# B&R Automation Studio project 8238 (part 5)

#### custom.st
```iecst
PROGRAM _INIT

	Std.TestMode;

//	FOR n := 1 TO MAX_CONTACTRON DO
//		incline						ACCESS ADR(IO_Link.Contactron[n]);
//		incline.Cmd.Reset_Automatic		:= 1;
//		tripCurrent						:= CONTACTRON_TRIP_50_PERCENT;
//		//tripCurrent						:= CONTACTRON_TRIP_75_PERCENT;
//	END_FOR;
//
//	camera ACCESS ADR(Camera[1].Interface);
//
//	gSettings.Drive[1].MotorSize	 			:= ABB_MOTOR_0_75KW;
//	gSettings.Drive[2].MotorSize	 			:= ABB_MOTOR_0_75KW;
//	gSettings.Drive[3].MotorSize	 			:= ABB_MOTOR_3KW;
//	gSettings.Drive[4].MotorSize	 			:= ABB_MOTOR_3KW;
////	gSettings.Drive[3].MotorSize	 			:= ABB_MOTOR_CUSTOM; //from motor template
//
//	FOR n := 1 TO MAX_DRIVES DO
//		ABB_EPL.Drives[n].Cmd.Direction 		:= ABB_DIRECTION_FWD;
//		ABB_EPL.Drives[n].Cmd.TargetVelocity 	:= gSettings.Drive[n].TargetVelocity;
//		gSettings.Drive[n].AccTime 				:= 0.5;
//		gSettings.Drive[n].DecTime 				:= 0.2;
//		gSettings.Drive[n].BrakeFitted			:= 0;
//	END_FOR;

END_PROGRAM

PROGRAM _CYCLIC

//	//==============================
//	//Inclines
//	//==============================
//
//	FOR n := 1 TO MAX_CONTACTRON DO
//		incline					ACCESS ADR(IO_Link.Contactron[n]);
//		IF 	(incline.Comms.Read.CurrentStatus = 0) THEN
//			incline.Cmd.Current		:= tripCurrent;
//		END_IF;
//	END_FOR;
//
//	IO_Link.Contactron[1].Cmd.Run := r57.run_slant; //SICU1		//Y[1399].Y06
//	IO_Link.Contactron[2].Cmd.Run := r116.run_slant; //CICU1
//	IO_Link.Contactron[3].Cmd.Run := r101.run_slant; //CICU2
//	IO_Link.Contactron[4].Cmd.Run := r127.run_slant; //CICU3
////	IO_Link.Contactron[2].Cmd.Run := r21.run_slant; //CICU4
//
//	//====================================
//	//TRN Controls
//	//====================================
//
//	//STRN2
//	r62.request_rotate := (r25.state = 1) AND (OpcUa.VC[232].Read.PositionNo = 2) AND (OpcUa.VC[232].Read.Auto) AND (OpcUa.VC[232].Read.ReadyToReceive) AND NOT r25.safety_zone;
//	ton_rotated_strn2(IN:= (r62.sw_out_a AND r62.sw_out_b),PT := T#2s);
//	ton_straight_strn2(IN:= (r62.sw_in_a AND r62.sw_in_b),PT := T#2s);
//	r62.custom_bring_lock := ton_rotated_strn2.Q OR r62.front_a OR r62.front_b OR NOT r62.rail_mt;
//	rotate_r62 := ((r62.state >= 6) AND (r62.state <= 7)) OR (r62.state = 9);
//	straight_r62 := ((r62.state = 8) OR (r62.state = 1) OR (r62.state = 5));
//	r62.clamp := (rotate_r62 AND NOT ton_rotated_strn2.Q) OR (straight_r62 AND NOT ton_straight_strn2.Q);  // We have to fire this to unlock the rails so we can move them
//
//	r25.custom_bring_lock := NOT ton_rotated_strn2.Q;
//	//r63.custom_bring_lock := NOT ton_straight_strn2.Q;
//
//	//STRN1
//	r63.request_rotate := NOT r22.safety_zone;
//	ton_rotated_strn1(IN:= (r63.sw_out_a AND r63.sw_out_b),PT := T#2s);
//	ton_straight_strn1(IN:= (r63.sw_in_a AND r63.sw_in_b),PT := T#2s);
//	r63.custom_bring_lock := ton_rotated_strn2.Q OR r63.front_a OR r63.front_b OR NOT r63.rail_mt OR NOT ton_straight_strn2.Q;
//	rotate_r63 := ((r63.state >= 6) AND (r63.state <= 7)) OR (r63.state = 9);
//	straight_r63 := ((r63.state = 8) OR (r63.state = 1) OR (r63.state = 5));
//	r63.clamp := (rotate_r63 AND NOT ton_rotated_strn1.Q) OR (straight_r63 AND NOT ton_straight_strn1.Q);  // We have to fire this to unlock the rails so we can move them
//
//	r22.custom_bring_lock := NOT ton_rotated_strn1.Q;
//
//
//	//CTRN1
//	r135.request_rotate := (r65.state = 1) AND (OpcUa.VC[241].Read.PositionNo = 2) AND (OpcUa.VC[241].Read.Auto) AND (OpcUa.VC[241].Read.ReadyToReceive);
//	ton_rotated_ctrn1(IN:= (r135.sw_out_a AND r135.sw_out_b), PT := T#2s);
//	ton_straight_ctrn1(IN:= (r135.sw_in_a AND r135.sw_in_b), PT := T#2s);
//	r135.custom_bring_lock := ton_rotated_ctrn1.Q OR r135.front_a OR r135.front_b OR NOT r135.rail_mt;
//	rotate_r135 := ((r135.state >= 6) AND (r135.state <= 7)) OR (r135.state = 9);
//	straight_r135 := ((r135.state = 8) OR (r135.state = 1) OR (r135.state = 5));
//	r135.clamp := (rotate_r135 AND NOT ton_rotated_ctrn1.Q) OR (straight_r135 AND NOT ton_straight_ctrn1.Q);  // We have to fire this to unlock the rails so we can move them
//
//	//CTRN2
//	r133.request_rotate := (r68.state = 1) AND (OpcUa.VC[242].Read.PositionNo = 2) AND (OpcUa.VC[242].Read.Auto) AND (OpcUa.VC[242].Read.ReadyToReceive);
//	ton_rotated_ctrn2(IN:= (r133.sw_out_a AND r133.sw_out_b), PT := T#2s);
//	ton_straight_ctrn2(IN:= (r133.sw_in_a AND r133.sw_in_b), PT := T#2s);
//	r133.custom_bring_lock := ton_rotated_ctrn2.Q OR r133.front_a OR r133.front_b OR NOT r133.rail_mt;
//	rotate_r133 := ((r133.state >= 6) AND (r133.state <= 7)) OR (r133.state = 9);
//	straight_r133 := ((r133.state = 8) OR (r133.state = 1) OR (r133.state = 5));
//	r133.clamp := (rotate_r133 AND NOT ton_rotated_ctrn2.Q) OR (straight_r133 AND NOT ton_straight_ctrn2.Q);  // We have to fire this to unlock the rails so we can move them
//
//
////	//====================================
////	//TRF Controls
////	//====================================
////
////	ton_clear_strf1(IN:= (NOT r22.front_a AND NOT r22.front_b),PT := T#2s);
////	ton_clear_strf2(IN:= (NOT r25.front_a AND NOT r25.front_b),PT := T#2s);
////
////	r63.custom_send_lock	:=	NOT ton_clear_strf1.Q AND (r22.state >= 5);
////	r62.custom_send_lock	:=	NOT ton_clear_strf2.Q AND (r25.state >= 5);
//
////==============================
////Custom for CDC6 & CDC7
////==============================
//	RequestBag 		:= WORD_TO_INT(plc_info1);
//	IF RequestBag = 7 THEN
//		cdc7RequestBag := TRUE;
//		cdc6RequestBag := FALSE;
//	ELSIF RequestBag = 6 THEN
//		cdc6RequestBag := TRUE;
//		cdc7RequestBag := FALSE;
//	ELSE
//		cdc6RequestBag := FALSE;
//		cdc7RequestBag := FALSE;
//	END_IF;
//
//	r104.lift_stp := r106.going_to;
//
//	// Clean custom code
//	r104.custom_bring_lock := cdc7RequestBag OR r106.going_to;
//	r106.custom_bring_lock := r104.going_to OR r104.front_raw OR NOT r104.rail_mt OR r104.fire;
//
//	r104.going_to;
//	r106.going_to;
//	r103.custom_send_lock;
////==============================
////Sorting Stations Mapping
////==============================
//
////	r41.jogmode := 1;	//set belt pulse mode = TRUE
////	r42.jogmode := 1;
////	r43.jogmode := 1;
////	r44.jogmode := 1;
////	r45.jogmode := 1;
////	r46.jogmode := 1;
////	r47.jogmode := 1;
////	r48.jogmode := 1;
////	r49.jogmode := 1;
////	r50.jogmode := 1;
//
//	//	IO_Link.Contactron[2].Cmd.Run := r41.run_conveyor AND (r40.conveyor_running OR (r40.run_conveyor AND Std.TestMode));
//	//	IO_Link.Contactron[3].Cmd.Run := r42.run_conveyor AND (r40.conveyor_running OR (r40.run_conveyor AND Std.TestMode));
//	//	IO_Link.Contactron[4].Cmd.Run := r43.run_conveyor AND (r40.conveyor_running OR (r40.run_conveyor AND Std.TestMode));
//	//	IO_Link.Contactron[5].Cmd.Run := r44.run_conveyor AND (r40.conveyor_running OR (r40.run_conveyor AND Std.TestMode));
//	//	IO_Link.Contactron[6].Cmd.Run := r45.run_conveyor AND (r40.conveyor_running OR (r40.run_conveyor AND Std.TestMode));
//	//	IO_Link.Contactron[7].Cmd.Run := r46.run_conveyor AND (r40.conveyor_running OR (r40.run_conveyor AND Std.TestMode));
//	//	IO_Link.Contactron[8].Cmd.Run := r47.run_conveyor AND (r40.conveyor_running OR (r40.run_conveyor AND Std.TestMode));
//	//	IO_Link.Contactron[9].Cmd.Run := r48.run_conveyor AND (r40.conveyor_running OR (r40.run_conveyor AND Std.TestMode));
//	//	IO_Link.Contactron[10].Cmd.Run := r49.run_conveyor AND (r40.conveyor_running OR (r40.run_conveyor AND Std.TestMode));
//	//	IO_Link.Contactron[11].Cmd.Run := r50.run_conveyor AND (r40.conveyor_running OR (r40.run_conveyor AND Std.TestMode));
//	//
//	r1.custom_send_lock := r1.over_weight;
//	r2.custom_send_lock := r2.over_weight;
//	r3.custom_send_lock := r3.over_weight;
//	r4.custom_send_lock := r4.over_weight;
//	r5.custom_send_lock := r5.over_weight;
//	r6.custom_send_lock := r6.over_weight;
//	r7.custom_send_lock := r7.over_weight;
//	r8.custom_send_lock := r8.over_weight;
//	r9.custom_send_lock := r9.over_weight;
//	r10.custom_send_lock := r10.over_weight;
//	r11.custom_send_lock := r11.over_weight;
//	r12.custom_send_lock := r12.over_weight;
//	r13.custom_send_lock := r13.over_weight;
//	r14.custom_send_lock := r14.over_weight;
//	r15.custom_send_lock := r15.over_weight;
//	r16.custom_send_lock := r16.over_weight;
//	r17.custom_send_lock := r17.over_weight;
//	r18.custom_send_lock := r18.over_weight;
//	r19.custom_send_lock := r19.over_weight;
//	r20.custom_send_lock := r20.over_weight;
//
//	//==============================
//	//Speed Reducers
//	//==============================
//
//	////////////////////////SSR1 is a brush style//////////////////////////
//
//	//inputs
//	i_bagApproach[1] := ssr1_prs; //ssr1 on soiled system
//	//i_bagApproach[2] := ssr2_prs; //ssr2 on soiled system
//	//i_bagApproach[3] := csr1_prs; //csr1 on clean system
//
//	FOR n := 1 TO MAX_SPEED_REDUCERS DO
//
//		ctu_tripCount[n](CU := i_bagApproach[n],PV := 2,RESET := ton_10ms_openBrush[n].Q);
//		ton_10ms_openBrush[n](IN := NOT SafetyZone[1].HaltSys AND o_closeBrush[n], PT := 300);
//
//		IF (ctu_tripCount[n].CV >= 2) THEN
//			o_closeBrush[n] := TRUE;
//		END_IF;
//
//		IF ton_10ms_openBrush[n].Q THEN
//			o_closeBrush[n] := FALSE;
//		END_IF;
//	END_FOR;
//
//	//Outputs
//	ssr1_close := o_closeBrush[1];
////	ssr2_close := o_closeBrush[2];
////	csr1_close := o_closeBrush[3];
//
//
//
//	//==============================
//	//ABB DRIVES
//	//==============================
//
//	FOR n := 1 TO MAX_DRIVES DO
//		ABB_EPL.Drives[n].Cmd.TargetVelocity := gSettings.Drive[n].TargetVelocity;
//	END_FOR;
//
//	ABB_EPL.Drives[1].Cmd.QuickStop := NOT SafetyZone[1].HaltSys; //SB1
//	ABB_EPL.Drives[2].Cmd.QuickStop := NOT SafetyZone[1].HaltSys; //SB2
//	ABB_EPL.Drives[3].Cmd.QuickStop := NOT SafetyZone[4].HaltSys; //STB1
//	ABB_EPL.Drives[4].Cmd.QuickStop := NOT SafetyZone[5].HaltSys; //STB2
//
////	tof_largeload(IN := X[1351].X06, PT:=t#10s);
////	IF tof_largeload.Q THEN
////		ABB_EPL.Drives[2].Cmd.TargetVelocity := gSettings.Drive[2].TargetVelocity/2;
////		//testspeed := gSettings.Drive[2].TargetVelocity/2;
////	ELSE
////		ABB_EPL.Drives[2].Cmd.TargetVelocity := gSettings.Drive[2].TargetVelocity;
////		//testspeed := gSettings.Drive[2].TargetVelocity;
////	END_IF;
//
//	//==============================
//	//SB1 & SB2 - PB control
//	//==============================
//	IF EDGENEG (sb1_start) THEN
//		runBelts_SB1 := 1;
//	END_IF;
//	IF NOT sb1_stop OR SafetyZone[1].HaltSys THEN
//		runBelts_SB1 := 0;
//	END_IF;
//
//	IF EDGENEG (sb2_start) THEN
//		runBelts_SB2 := 1;
//	END_IF;
//	IF NOT sb2_stop OR SafetyZone[1].HaltSys THEN
//		runBelts_SB2 := 0;
//	END_IF;
//
//	sb1_lamp := runBelts_SB1;
//	sb2_lamp := runBelts_SB2;
//
//	ABB_EPL.Drives[1].Cmd.Run := (runBelts_SB1) AND sb1_endPX;
//	ABB_EPL.Drives[2].Cmd.Run := (runBelts_SB2) AND sb2_endPX;
//	ABB_EPL.Drives[3].Cmd.Run := r21.run_conveyor;
//	r21.conveyor_running := ABB_EPL.Drives[3].Status.Running OR r21.run_conveyor;
//	ABB_EPL.Drives[4].Cmd.Run := r24.run_conveyor;
//	r24.conveyor_running := ABB_EPL.Drives[4].Status.Running OR r24.run_conveyor;
//
//
//	//==============================
//	//UI Indicators - in iolist
//	//==============================
//
//
//
//	//==============================
//	//Timers
//	//==============================
//
//	SetValueByName('R043','DBNC_after_time',50);
//	SetValueByName('R045','DBNC_after_time',50);
//	SetValueByName('R047','DBNC_after_time',50);
//	SetValueByName('R092','DBNC_after_time',50);
////	SetValueByName('R047','DBNC_after_time',50);
////	SetValueByName('R047','DBNC_after_time',50);
//	//	SetValueByName('R042','PulseTimerOffTime',1000);
////	//SetValueByName('R043','PulseTimerOnTime',3000);
////	SetValueByName('R043','PulseTimerOffTime',1000);
////	//SetValueByName('R044','PulseTimerOnTime',3000);
////	SetValueByName('R044','PulseTimerOffTime',1000);
////	//SetValueByName('R045','PulseTimerOnTime',3000);
////	SetValueByName('R045','PulseTimerOffTime',1000);
////	//SetValueByName('R046','PulseTimerOnTime',3000);
////	SetValueByName('R046','PulseTimerOffTime',1000);
////	//SetValueByName('R047','PulseTimerOnTime',3000);
////	SetValueByName('R047','PulseTimerOffTime',1000);
////	//SetValueByName('R048','PulseTimerOnTime',3000);
////	SetValueByName('R048','PulseTimerOffTime',1000);
////	//SetValueByName('R049','PulseTimerOnTime',3000);
////	SetValueByName('R049','PulseTimerOffTime',1000);
////	//SetValueByName('R050','PulseTimerOnTime',3000);
////	SetValueByName('R050','PulseTimerOffTime',1000);
////	//SetValueByName('R041','PulseTimerOnTime',3000);
////	//SetValueByName('R041','PulseTimerOffTime',5000);
////	//SetValueByName('R040','MaximumRunningTime',200000);
////	//	SetValueByName('R041','DBNC_front_time',2000);
////	//	SetValueByName('R076','DBNC_front_time',1000);
////	//
////
////	// Camera
////	camera.Read := r31.front;
////	IF camera.ResultReady AND r31.front THEN
////		brsmemcpy(ADR(barcode1),ADR(camera.Result),SIZEOF(barcode1));
////	ELSE
////		brsmemset(ADR(barcode1),0,SIZEOF(barcode1));
////	END_IF;
////
////	IF EDGEPOS(camera.Read) THEN
////		readCount := readCount + 1;
////	END_IF;
////
////
////	//
////	tof_cameraClean(IN := (readCount > 100), PT:=t#2s);
////	r31.puncher := NOT tof_cameraClean.Q;
////
////	IF (readCount > 105) THEN
////		readCount := 0;
////	END_IF;

END_PROGRAM
```

#### Variables.var
```iecst
VAR
	incline : REFERENCE TO Contactron_Type;
	ton_settled : TON_10ms;
	ton_tiltDown : TON_10ms;
	ton_tiltUp : TON_10ms;
	ton_CloserDown : TON_10ms;
	ton_CloserUp : TON_10ms;
	tilt : USINT;
	ton_WaitExtendArm : TON_10ms;
	n : USINT;
	recircLoad : BOOL;
	runBelts : BOOL;
	CarousalBlockedTime : UDINT;
	CarousalBlockedTimer : TON_10ms;
	tof_pressure_1 : TOF;
	tof_open_pressure_1 : TOF;
	camera : REFERENCE TO Camera_interface_typ;
	testing : BOOL;
	testweight1 : UINT;
	testweight2 : UINT;
	runBelts_SB1 : BOOL;
	runBelts_SB2 : BOOL;
	tof_cameraClean : TOF;
	readCount : UINT;
	r81_clear_timer : TON;
	clear_time : UDINT := 5000;
	tof_pressureTime : UDINT := 3000;
	tof_pressureTime2 : UDINT := 1000;
	ctu_tripCount : ARRAY[0..MAX_SPEED_REDUCERS] OF CTU;
	i_bagApproach : ARRAY[0..MAX_SPEED_REDUCERS] OF BOOL;
	ton_10ms_countDebounce : ARRAY[0..MAX_STATIONS] OF TON_10ms;
	ton_10ms_openBrush : ARRAY[0..MAX_SPEED_REDUCERS] OF TON_10ms;
	o_closeBrush : ARRAY[0..MAX_SPEED_REDUCERS] OF BOOL;
	lowerGuard : BOOL;
	tof_largeload : TOF;
	testspeed : INT;
	ton_rotated_strn1 : TON;
	ton_straight_strn1 : TON;
	ton_rotated_strn2 : TON;
	ton_straight_strn2 : TON;
	ton_clear_strf1 : TON;
	ton_clear_strf2 : TON;
	rotate_r62 : BOOL;
	straight_r62 : BOOL;
	rotate_r63 : BOOL;
	straight_r63 : BOOL;
	ton_rotated_ctrn1 : TON;
	ton_straight_ctrn1 : TON;
	ton_rotated_ctrn2 : TON;
	ton_straight_ctrn2 : TON;
	ton_clear_ctrf1 : TON;
	ton_clear_ctrf2 : TON;
	rotate_r135 : BOOL;
	straight_r135 : BOOL;
	rotate_r133 : BOOL;
	straight_r133 : BOOL;
	RequestBag : INT;
	countMode : BOOL;
	iCount : ARRAY[0..MAX_STATIONS] OF BOOL;
	cntDebounceLatch : ARRAY[0..MAX_STATIONS] OF BOOL;
END_VAR
```

#### LocalFunctions.fun
```iecst
{REDUND_ERROR} FUNCTION SetValueByName : BOOL (**Set Local variable from external task*) (*$GROUP=User,$CAT=User,$GROUPICON=User.png,$CATICON=User.png*)
	VAR_INPUT
		TaskName : STRING[24];
		VarName : STRING[50];
		Value : UDINT;
	END_VAR
	VAR
		sVar : UDINT;
		pVar : UDINT;
		varName : STRING[75];
	END_VAR
END_FUNCTION
```

#### SetValueByName.st
```iecst
//*Set Local variable from external task
FUNCTION SetValueByName
	SetValueByName := 0;
	varName := '::';
	brsstrcat(ADR(varName),ADR(TaskName));
	brsstrcat(ADR(varName),ADR(':'));
	brsstrcat(ADR(varName),ADR(VarName));

	IF (PV_xgetadr(ADR(varName),ADR(pVar),ADR(sVar)) = 0) THEN
		IF (SIZEOF(Value) <= sVar)THEN
			brsmemcpy(pVar,ADR(Value),SIZEOF(Value));
			SetValueByName := 1;
		ELSE
			brsmemcpy(pVar,ADR(Value),sVar);
			SetValueByName := 1;
		END_IF;
	END_IF;
END_FUNCTION
```

- Visualisation Logical/mappView (not shown)

### SystemConstants.var - *SYSTEM Constants
```iecst
VAR CONSTANT
	MAX_CAMERAS : USINT := 1; (** Number of B&R Barcode scanners*)
	MAX_SPEED_REDUCERS : USINT := 1; (*Set to number of speed reducers*)
	MAX_CONTACTRON : USINT := 4;
	MAX_DRIVES : USINT := 16; (*Set to number of drives*)
	MAX_FUSE_BANKS : USINT := 11;
	MAX_DUAL_CHANNELS : USINT := 10; (** Number of Estops*)
	MAX_HOIST : USINT := 4;
	MAX_SAFE_ZONES : USINT := 30;
	MAX_RAILS : UINT := 136; (**DO NOT USE -> USE RAIL_COUNT INSTEAD*)
END_VAR
```

### Program Logical/Standard/Program (IEC) - * PLAY AREA

#### Variables.var
```iecst
VAR
	myBuffer : ARRAY[0..511] OF INT;
	myAsIoTrcGet : AsIoTrcGet;
	mO_info : MO_info;
	test : UINT;
	datObjCreate : DatObjCreate;
	FileCreate_0 : FileCreate;
	FileInfo_0 : FileInfo;
	FileOpen_0 : FileOpen;
	ident : UDINT;
	Path : STRING[80];
	fileRW : fileReadWrite;
	sysFileName : STRING[10];
	getModuleName : GetModuleName;
	moduleAddress : STRING[30];
	testUsint : USINT;
END_VAR
```

#### Main.st
```iecst
PROGRAM _INIT
	(* Insert code here *)
	Path := 'SL1.IF1.ST11.IF1.ST3.TRC';
	myAsIoTrcGet.pDevice := ADR(Path);//'SS1.IF1.ST131.TRC');
	myAsIoTrcGet.pBuffer := ADR(myBuffer);
	myAsIoTrcGet.bufferLen := SIZEOF(myBuffer);
	//Sys file to try
//	User			XML - Users
//	Role			XML - Roles
//	sysconf			NOT AVAILABLE ?
//	ashwd			NOT READABLE
//	arconfig		XML -- Contains all hardware configuration  !!! Use this to get module name. ***
//	asfw			NOT READABLE
//	ashwac			XML -- No data ??
//	iomap			IO File - Readable
//	asiol1			XML -- No data ??
//	asiol3			XML -- No data ??
//	Config			XML -- MAPP Components config
//	TC				XML -- Text Config.
//	viComp			VISION
//	Settings		VISION
//	viAppBCDE		VISION

	sysFileName := 'iomap';
END_PROGRAM

PROGRAM _CYCLIC

	//We can run an IO trace.. Is this useful when looking for breaks in the IO.. Maybe we can run somekind of automated test.

	IF myAsIoTrcGet.enable <> 0 THEN
		myAsIoTrcGet();
		myAsIoTrcGet.enable := 0;
	END_IF

	// Testing resolving the Module Name.

	CASE test OF
		10:

			mO_info(enable := 1, pName := ADR(sysFileName), grp := 0);
			IF mO_info.status = ERR_OK THEN
				test := 20;
			END_IF;

		20:// File Write
			fileRW.enable := 1;
			fileRW.mode := FILE_SAVE;
			fileRW.pData := mO_info.address;
			fileRW.sizeData := 	mO_info.size;
			fileRW.pFileDevice := ADR('user');
			fileRW.pFileName := ADR(sysFileName);
			fileRW();
			IF fileRW.status = ERR_OK THEN
				test := 0;
			ELSIF fileRW.status <> ERR_FUB_BUSY THEN
				test := 100;
			END_IF;

		50:// Read a module name
			getModuleName.enable := 1;
			getModuleName.pModuleAddress := ADR(moduleAddress);
			getModuleName();
			IF getModuleName.status = ERR_OK THEN
				test := 0;
			ELSIF (getModuleName.status <> ERR_FUB_BUSY) THEN
				test := 100;
			END_IF;

	END_CASE;

END_PROGRAM

PROGRAM _EXIT
	(* Insert code here *)

END_PROGRAM
```

### Constants_ABB.var - Exported constants
```iecst
(*Insert your comment here.*)
VAR CONSTANT
	MAX_PARAMS : USINT := 20; (*Maximum number of params*)
END_VAR
(**Controls*)
VAR
	ABB_MAX_VELOCITY : {REDUND_UNREPLICABLE} INT := 60; (*Maximum Frequency Allowed in hz*)
	ABB_MIN_VELOCITY : {REDUND_UNREPLICABLE} INT := 20; (*Minimum allowable speed of the drive*)
END_VAR
```

### ABB_EPL.var
```iecst
VAR
	ABB_EPL : ABB_EPL_Struct;
END_VAR
(*ALARM CODE*)
VAR CONSTANT
	ABB_FAULT_STO : UINT := 16#A5A0;
END_VAR
```

### ABB_EPL.typ
```iecst
TYPE
	ABB_EPL_Struct : 	STRUCT
		Drives : ARRAY[1..MAX_DRIVES]OF ABB_EPL_typ;
	END_STRUCT;
	ABB_EPL_typ : 	STRUCT
		Comm : ABB_EPL_Comm_typ;
		Cmd : ABB_EPL_cmd_typ;
		Status : ABB_EPL_status_typ;
		Config : EPL_Config;
		Manual : ABB_Manual_typ;
	END_STRUCT;
	ABB_EPL_Comm_typ : 	STRUCT
		ControlWord : UINT;
		StatusWord : UINT;
		ModuleOk : BOOL;
		State : ABB_EPL_Comm_State_enum;
		TargetVelocity : INT; (*RPM*)
		ActVelocity : INT; (*RPM*)
		ActCurrent : DINT;
		ActTorque : DINT;
		ErrorCode : UINT;
	END_STRUCT;
	ABB_Motor_Size_enum :
		(
		ABB_MOTOR_0_25KW := 0,
		ABB_MOTOR_0_37KW_0_91A_1374 := 1,
		ABB_MOTOR_0_37KW_0_97A_1342 := 2,
		ABB_MOTOR_0_37KW_1_14A_1380 := 3,
		ABB_MOTOR_0_75KW := 4,
		ABB_MOTOR_1_5KW := 5,
		ABB_MOTOR_2_2KW_4_75A_1450 := 6,
		ABB_MOTOR_3KW := 7,
		ABB_MOTOR_CUSTOM := 8
		);
	ABB_EPL_cmd_typ : 	STRUCT
		TargetVelocity : INT; (*RPM*)
		Run : BOOL;
		Reset : BOOL;
		QuickStop : BOOL;
		Direction : ABB_DIRECTION_Enum;
	END_STRUCT;
	ABB_EPL_Comm_State_enum :
		(
		ABB_DISCONNECTED := 0,
		ABB_QUICK_STOP := 1,
		ABB_CONFIG := 2,
		ABB_SWITCH_ON_INHIBITED := 3,
		ABB_NOT_READY_TO_SWITCH_ON := 4,
		ABB_READY_TO_SWITCH_ON := 5,
		ABB_READY_TO_RUN := 6,
		ABB_RUNNING := 7,
		ABB_TRIPPED := 8,
		ABB_OFF_REMOTE := 9, (**Drive not on remote control*)
		ABB_STO := 10,
		ABB_RAMP_DOWN := 11,
		ABB_INIT := 12 (*Driver is init*)
		);
	ABB_EPL_status_typ : 	STRUCT
		ReadyToSwitchOn : BOOL;
		ReadyToRun : BOOL;
		Tripped : BOOL;
		DriveEnabled : BOOL;
		QuickstopActive : BOOL;
		SwitchOnInhibit : BOOL;
		Warning : BOOL;
		AtSpeed : BOOL; (**Drive is running at target velocity*)
		ActCurrent : DINT; (*Amps*)
		ActTorque : DINT; (*% of nominal motor torque*)
		ThermalTrip : BOOL;
		OnRemote : BOOL; (**Powerlink control is active*)
		Running : BOOL;
	END_STRUCT;
	ABB_DIRECTION_Enum :
		(
		ABB_DIRECTION_FWD := 0,
		ABB_DIRECTION_REV := 1
		);
	EPL_Config : 	STRUCT
		function : EplSDOWrite;
		currentParam : USINT;
		params : ARRAY[0..MAX_PARAMS]OF EPL_SDO;
		Node : USINT;
		EPL_Address : STRING[25];
	END_STRUCT;
	ABB_Manual_typ : 	STRUCT
		Enable : BOOL; (*Visu Index for Manual Control*)
		Run : BOOL;
		Velocity : INT;
		Direction : ABB_DIRECTION_Enum;
		ErrorReset : BOOL;
	END_STRUCT;
	EPL_SDO : 	STRUCT
		index : UINT;
		subIndex : USINT;
		data : DINT;
		datalen : UDINT;
		status : UINT;
		errorInfo : UDINT;
	END_STRUCT;
	ABB_Settings_typ : 	STRUCT  (**Moved to gSettings Structure*)
		MotorSize : ABB_Motor_Size_enum;
		BrakeFitted : BOOL; (*Does the motor have a brake fitted*)
		AccTime : REAL;
		DecTime : REAL;
		AutoReset : BOOL := 0; (**Option to auto reset errors.*)
		Name : STRING[50];
		TargetVelocity : INT;
	END_STRUCT;
END_TYPE
```

### Program Logical/Standard/ABB_EPL/ABB_Driver (IEC, version 4.00.4)

#### ControlWord.var - Exported constants
```iecst
(*CONTROL WORD STATES- DO NOT CHANGE*)
VAR CONSTANT
	DISABLE_VOLTAGE : UINT := 2#0000010000000000; (*Constanst for setting control word in case statement*)
	FAULT_RESET : UINT := 2#0000010011110000; (*Constanst for setting control word in case statement*)
	QUICK_STOP : UINT := 2#0000010001110000; (*Constanst for setting control word in case statement*)
	ENABLE_OPERATION : UINT := 2#0000010001111111; (*Constanst for setting control word in case statement*)
	RAMP_DOWN : UINT := 2#0000010001110111; (*Constanst for setting control word in case statement*)
	SHUT_DOWN : UINT := 2#0000010001110110; (*Constanst for setting control word in case statement*)
	SET_REMOTE : UINT := 2#0000010000000000; (*Constanst for setting control word in case statement*)
	SWITCH_ON : UINT := 2#0000010001110111; (*Constanst for setting control word in case statement*)
END_VAR
```

#### Main.st - Init, cyclic, exit code
```iecst
//V2.00.1 -- First stable release
//V2.00.2 -- Set brake control to be optional - This means changing when we encode the paramater structure.
//V2.00.3 -- Add new constant to set MAX_FREQUENCY
//V2.00.4 -- If the drive started not on remote it wouldn;t always go into config to start. ADD new mode for when module ok is false.
//V2.00.5 -- Add test mode for simulation
//V2.00.6 -- BUG FIX -- Minumum speed was being set to Max which stopped speed control
//V2.00.7 -- REMOVE -- Remove the old structure for settings via http
//V2.00.8 -- FIX -- Correct the scaling of MaxCurrent from settings - we now us 200 = 2A
//V3.00.1 -- CHANGE Combine Settings task into driver- Remove parameters from EPL write and move to SDO configuration function block
//V3.00.2 -- ADD Manual control mode via http!
//V3.00.3 -- Convert Manual Control to mappView.
//V4.00.1 -- Automatically get node number from PV structure.
//V4.00.2 -- Move Control word states into the program as the were not being copy when the task was moved causing errors.
//V4.00.3 -- Change halt mode of belts to we do a proper decel
//V4.00.4 -- Change error handling to always reset STO automatically

PROGRAM _INIT
	setNodeNumber.pDevice := ADR('SL1.IF1');
	FOR n := 1 TO MAX_DRIVES DO
		drive ACCESS ADR(ABB_EPL.Drives[n]);
		drive.Comm.State := ABB_CONFIG;
		drive.Config.currentParam := 1; //Reset starting parameter index
		drive.Config.Node := 0;
		drive.Config.EPL_Address := '';
		index := 0;
		init_state := 0;
	END_FOR;

	FOR n := 1 TO 8 DO
		visu_manual[n].ListBoxVisible := 0;
		visu_manual[n].TargetVelocity := ABB_MIN_VELOCITY;
		visu_manual[n].selectedIndex := 0;
	END_FOR;

	IF (MAX_DRIVES > 8) THEN
		max_manualControls := 8;
	ELSIF (MAX_DRIVES > 1) THEN
		max_manualControls := MAX_DRIVES;
	ELSE
		max_manualControls := 1;
	END_IF;
	xRun := FALSE;
END_PROGRAM

PROGRAM _CYCLIC

	IF EDGENEG(xRun) THEN
		FOR n := 1 TO MAX_DRIVES DO
			drive ACCESS ADR(ABB_EPL.Drives[n]);
			drive.Comm.State := ABB_INIT;
			drive.Config.currentParam := 1; //Reset starting parameter index
			drive.Config.Node := 0;
			drive.Config.EPL_Address := '';
			index := 0;
			init_state := 0;
		END_FOR;
	ELSIF NOT xRun THEN
		_getNodeInfo;
	ELSE

		_manual;  // mappView manual control.
		FOR x := 1 TO MAX_DRIVES DO
			IF (testDrive > 0) THEN
				n := testDrive;
			ELSE
				n := x;
			END_IF;

			drive 		ACCESS ADR(ABB_EPL.Drives[n]);
			settings	ACCESS ADR(gSettings.Drive[n]);

			//Control Word												Status Word
			//Bit 0		Switch On										Bit 0	Ready To Switch On
			//Bit 1		Enable Voltage									Bit 1	Switched On
			//Bit 2		Quick Stop										Bit 2	Operation Enabled
			//Bit 3		Enable Operation								Bit 3	Fault
			//Bit 4		Not Used In Scalor Mode							Bit 4	Voltage Enabled
			//Bit 5		Not Used In Scalor Mode							Bit 5	Quick Stop
			//Bit 6		Not Used In Scalor Mode							Bit 6	Switch On Disabled
			//Bit 7		Fault Reset										Bit 7 	Warning
			//Bit 8		Halt											Bit 8	Drive Specific TBC
			//Bit 9		Operation Mode Specific							Bit 9	Remote
			//Bit 10	Reserved	??Remote Control??					Bit 10	Target Reached
			//Bit 11	Drive Specific	TBC								Bit 11 	Internal Limit Reached
			//Bit 12	Drive Specific	TBC								Bit 12	Not Used In Scalor Mode
			//Bit 13	Drive Specific	TBC								Bit 13	Not Used In Scalor Mode
			//Bit 14	Drive Specific	TBC								Bit 14	Drive Specific TBC
			//Bit 15	Drive Specific	TBC								Bit 15	Drive Specific TBC

			//Use a local instance of controlword so we don't pass changing data to the drive while processing

			controlWord := SHUT_DOWN;	// 0000 0000 0111 0110

			//Encode the controlword and statusword
			_packData;

			IF Std.TestMode AND NOT drive.Comm.ModuleOk THEN // TEST MODE
				IF drive.Cmd.Run THEN
					drive.Comm.State := ABB_RUNNING;
				ELSE
					drive.Status.ReadyToRun := 1;
				END_IF;
			ELSIF NOT drive.Comm.ModuleOk THEN
				drive.Comm.State := ABB_DISCONNECTED;
			ELSIF (drive.Config.params[MAX_PARAMS].status <> 0) OR (drive.Config.currentParam < MAX_PARAMS) THEN
				drive.Comm.State := ABB_CONFIG;
			ELSIF NOT drive.Status.OnRemote THEN
				drive.Comm.State := ABB_OFF_REMOTE;
			ELSIF drive.Status.Tripped THEN
				drive.Comm.State := ABB_TRIPPED;
			ELSIF NOT drive.Cmd.QuickStop THEN	//Enable quick stop
				drive.Comm.State := ABB_QUICK_STOP;
			ELSIF drive.Status.SwitchOnInhibit THEN
				drive.Comm.State := ABB_SWITCH_ON_INHIBITED;
			ELSIF drive.Comm.ErrorCode = ABB_FAULT_STO THEN
				drive.Comm.State := ABB_STO;
			END_IF;

			CASE drive.Comm.State OF

				ABB_DISCONNECTED:
					drive.Config.currentParam := 1; // Force write of parameters

				ABB_CONFIG: //Wait for module OK to be TRUE
					_setParameters; //Write params
					IF drive.Comm.ModuleOk AND (drive.Config.params[MAX_PARAMS].status = 0) THEN
						drive.Comm.State := ABB_SWITCH_ON_INHIBITED;
					END_IF;

				ABB_SWITCH_ON_INHIBITED:	//Wait for quick stop and enable to be true
					IF NOT drive.Status.SwitchOnInhibit THEN
						drive.Comm.State := ABB_NOT_READY_TO_SWITCH_ON;
					END_IF;

				ABB_NOT_READY_TO_SWITCH_ON:
					IF drive.Status.ReadyToSwitchOn THEN
						drive.Comm.State := ABB_READY_TO_SWITCH_ON;
					END_IF;

				ABB_READY_TO_SWITCH_ON:
					controlWord := SWITCH_ON; //0000 0111 0111
					IF drive.Status.ReadyToRun THEN
						drive.Comm.State := ABB_READY_TO_RUN;
					END_IF;

				ABB_READY_TO_RUN:
					controlWord := SWITCH_ON; //0000 0111 0111
					IF drive.Cmd.Run AND (ABS(drive.Cmd.TargetVelocity) >= ABB_MIN_VELOCITY) AND NOT drive.Manual.Enable THEN //Check min frequency is met
						drive.Comm.State := ABB_RUNNING;
					ELSIF drive.Manual.Run AND (ABS(drive.Manual.Velocity) >= ABB_MIN_VELOCITY)  THEN
						drive.Comm.State := ABB_RUNNING;
					END_IF;

				ABB_RUNNING:
					controlWord := ENABLE_OPERATION; //0000 0111 1111
					IF NOT (drive.Cmd.Run AND NOT drive.Manual.Enable) AND NOT (drive.Manual.Run AND drive.Manual.Enable) THEN
						drive.Comm.State := ABB_RAMP_DOWN;
					END_IF;

				ABB_RAMP_DOWN:
					controlWord := RAMP_DOWN; //0001 0111 1111
					IF drive.Comm.StatusWord.11 = 0 AND drive.Comm.ActVelocity = 0 THEN
						drive.Comm.State := ABB_READY_TO_RUN;
					END_IF;

				ABB_QUICK_STOP:
					controlWord := QUICK_STOP; //0000 0111 0010
					IF drive.Comm.StatusWord.11 = 0 AND drive.Comm.ActVelocity = 0 AND drive.Cmd.QuickStop THEN
						drive.Comm.State := ABB_READY_TO_RUN;
					END_IF;

				ABB_TRIPPED: // AUTO Reseting -- We should change to manual reset..
					//We must wait for the drive to be ready for reset and give an edge.
						IF (drive.Comm.StatusWord.11 = 0) AND (drive.Comm.ActVelocity = 0) THEN
							IF settings.AutoReset THEN
								controlWord := FAULT_RESET;
							ELSIF drive.Manual.ErrorReset THEN
								controlWord := FAULT_RESET;
								drive.Manual.ErrorReset := FALSE; // Reset the command.
							ELSIF (drive.Comm.ErrorCode = 16#A5A0) THEN
								controlWord := FAULT_RESET; // ALWAYS CLEAR THE STO ERROR AUTO MATICALLY
							ELSIF (drive.Comm.ErrorCode = 0) THEN
								controlWord := FAULT_RESET; // THE FAULT HAS BEEN CLEARED EXTERNALLY
							END_IF;
						ELSE
							controlWord := DISABLE_VOLTAGE; //0000 0000 0000
						END_IF;

					//We can auto reset here..but we should log an error somewhere..
					IF NOT drive.Status.Tripped THEN
						drive.Manual.ErrorReset := FALSE; // Reset the command.
						drive.Cmd.Reset	 		:= FALSE;
						drive.Comm.State := ABB_SWITCH_ON_INHIBITED;
					END_IF;

				ABB_OFF_REMOTE:
					//Remote control not active
					controlWord := SET_REMOTE;
					////				IF drive.Status.OnRemote THEN
					////					IF (drive.Config.params[MAX_PARAMS].status <> 0) THEN
					////						drive.Comm.State := ABB_CONFIG;
					////					ELSE
					////						drive.Comm.State := ABB_SWITCH_ON_INHIBITED;
					////					END_IF;
					////				END_IF;
					//				IF NOT Std.Drives_AllowLocalMode AND (drive.Config.params[13].data = Std.Drives_AllowLocalMode) THEN //Only reset the parameters if the local control mode has chnaged
					//					_encodeParameters;
					//					drive.Config.currentParam := 1; //Reset starting parameter index
					//				END_IF;
					//
				ABB_STO:
					IF drive.Comm.ErrorCode <> ABB_FAULT_STO THEN
						drive.Comm.State := ABB_SWITCH_ON_INHIBITED;
					END_IF;

			END_CASE;
			drive.Status.Running := (drive.Comm.State =  ABB_RUNNING);
			drive.Comm.ControlWord := controlWord;

			drive.Manual := DRIVE_MANUAL_DEFAULT;
		END_FOR;

	END_IF;

	//Temp code so that we can set a node number, The NODE must already be set to 1 (DEFAULT)
	IF (newNode > 0) THEN
		setNodeNumber.enable := 1;
		setNodeNumber.node := 1;
		setNodeNumber.index := 16#4033;
		setNodeNumber.subindex := 16#03;
		setNodeNumber.pData :=  ADR(newNode);
		setNodeNumber.datalen := 2;
		setNodeNumber();
		IF (setNodeNumber.status = ERR_OK) THEN
			newNode := 0;
		END_IF;
	ELSIF saveNewNode THEN
		saveVar := 1;
		setNodeNumber.enable := 1;
		setNodeNumber.node := 1;
		setNodeNumber.index := 16#4033;
		setNodeNumber.subindex := 16#1B;
		setNodeNumber.pData :=  ADR(saveVar);
		setNodeNumber.datalen := 2;
		setNodeNumber();
		IF (setNodeNumber.status = ERR_OK) THEN
			saveNewNode := 0;
		END_IF;
	ELSIF (factoryReset > 0) THEN
		saveVar := 34560;
		setNodeNumber.enable := 1;
		setNodeNumber.node := UINT_TO_USINT(factoryReset);
		setNodeNumber.index := 16#4060;
		setNodeNumber.subindex := 16#06;
		setNodeNumber.pData :=  ADR(saveVar);
		setNodeNumber.datalen := 2;
		setNodeNumber();
		IF (setNodeNumber.status = ERR_OK) THEN
			factoryReset := 0;
		END_IF;
	END_IF;

END_PROGRAM
```

#### Types.typ - Local data types
```iecst
TYPE
	abb_visu_manual_typ : 	STRUCT
		Visible : BOOL; (**Are the controls Visible*)
		Name : STRING[50];
		Node : USINT;
		ModuleOk : BOOL;
		ActVelocity : INT; (*RPM*)
		ActCurrent : DINT;
		ActTorque : DINT;
		ErrorCode : UINT;
		RunReverse : BOOL;
		RunForwards : BOOL;
		State : STRING[40]; (**Text picker was being a pain in group box so print string output.*)
		TargetVelocity : INT;
		ErrorReset : BOOL;
		ErrorActive : BOOL;
		selectedIndex : UINT;
		selectedValue : STRING[10];
		refreshDropDown : R_TRIG;
		ListBoxVisible : BOOL;
		EnableRunReverse : BOOL;
		EnableRunForwards : BOOL;
	END_STRUCT;
END_TYPE
```

#### Variables.var - Local variables
```iecst
VAR
	drive : REFERENCE TO ABB_EPL_typ; (*ref var to drive structure*)
	controlWord : UINT; (*control word for drive*)
	n : USINT; (*used to hold loop state*)
	testDrive : USINT; (*set this to drive number you want to test*)
	i : USINT;
	count : USINT;
	test : UINT;
	newNode : UINT;
	saveNewNode : BOOL;
	saveVar : UINT;
	factoryReset : UINT;
	setNodeNumber : EplSDOWrite;
	nominalCurrent_9906 : DINT;
	nominalPower_9910 : DINT;
	nominalSpeed_9909 : DINT;
	maxCurrent : DINT;
	accTime : DINT;
	decTime : DINT;
	x : USINT;
	visu_man : REFERENCE TO abb_visu_manual_typ;
	visu_manual : ARRAY[0..8] OF abb_visu_manual_typ;
	index : UINT;
	xRun : BOOL;
	config : REFERENCE TO EPL_Config;
	pvName : STRING[30];
	getNode : getNodeFromPV;
	driveNo : STRING[5];
	settings : REFERENCE TO ABB_Settings_typ;
	init_state : USINT;
	sNode : STRING[5];
	moduleAddress : STRING[75];
	getModuleName : GetModuleName;
END_VAR
VAR CONSTANT
	DRIVE_MANUAL_DEFAULT : ABB_Manual_typ := (Enable:=0,Run:=0,Velocity:=0,Direction:=ABB_DIRECTION_FWD,ErrorReset:=0);
END_VAR
VAR
	manualSelectDrowDown : ARRAY[0..MAX_DRIVES] OF STRING[125]; (*JSON for the drop downs on manual mode.*)
	sIndex : STRING[5];
	updateDropDown : BOOL;
	selIndex : DINT;
	max_manualControls : USINT;
	targetSpeedValid : BOOL;
END_VAR
```

#### encodeParameters.st
```iecst
//-----------------------------------------
//--AsEPL library Status Error Codes-------
//-----------------------------------------

//Error									Description
//0  										No error
//65534  								Function block parameter "enable" not equal to 1
//65535  								Function block still working

//31340  								Basis of error numbers, internal error
//31341  								Specified device not a POWERLINK interface
//31342  								Function can only be executed on an MN (managing node).
//31343  								Function can only be executed on a CN (controlled node).
//31344  								Read or write access failed. See errorinfo for the precise cause of the error.
//31345  								Input parameters outside of permitted value range
//31346  								Specified index already exists
//31347  								Specified subindex already exists
//31348  								Specified index does not exist
//31349  								Specified subindex does not exist
//31392  								Null pointer given as data buffer
//31399  								Error code for non-implemented functionality

//-----------------------------------------
//-----AsEPL library Error Info Codes------
//-----------------------------------------

//Error									Description
//16#0504_0000 					SDO communication timeout.
//16#0504_0001 					Invalid or unknown client/server command.
//16#0504_0002 					Size of transferred data invalid.
//16#0504_0003 					Error in sequence layer.
//16#0504_0005 					Could not allocate enough memory.
//16#0601_0000 					Cannot access object.
//16#0601_0001 					Attempted to read a write-only object.
//16#0601_0002 					Attempted to write a read-only object.
//16#0602_0000 					Object not in object dictionary.
//16#0604_0041 					Attempted to map an object in the PDO that doesn't support it.
//16#0604_0042 					Assignment would exceed PDO length.
//16#0604_0043 					General parameter incompatibility.
//16#0604_0047 					General device incompatibility.
//16#0606_0000 					Access failed due to hardware error.
//16#0607_0010 					Data type doesn't match the length of the access.
//16#0607_0012 					Length of the access is larger than the length of the data type.
//16#0607_0013 					Length of the access is smaller than the length of the data type.
//16#0609_0011 					Subindex does not exist.
//16#0609_0030 					Invalid value range.
//16#0609_0031 					Value too high for value range.
//16#0609_0032 					Value too low for value range.
//16#0609_0036 					Maximum value less than minimum value.
//16#0800_0000 					General error.
//16#0800_0020 					Cannot transfer or store data.
//16#0800_0021 					Data cannot be transferred or stored since it's being used locally by the device.
//16#0800_0022 					Data cannot be transferred or saved due to the device state.

ACTION _encodeParameters:
	//Clear all parameters
	FOR i:= 1 TO MAX_PARAMS DO
		//Clear stauts/error
		drive.Config.params[i].status := 1; //Set to 1 here, if not cleared when written is shows it has not been written
		drive.Config.params[i].errorInfo := 0;
	END_FOR;

	//Set all parameters
	//Brake Function
	drive.Config.params[1].index := 16#402C;	//Brake Control Enable 44.06
	drive.Config.params[1].subIndex := 16#6;
	drive.Config.params[1].data := BOOL_TO_DINT(settings.BrakeFitted);	//Enable brake control
	drive.Config.params[1].datalen := 4;

	drive.Config.params[2].index := 16#400A;	//RO1 Source 10.24
	drive.Config.params[2].subIndex := 16#18;
	drive.Config.params[2].data := 22;	//Relay is active when brake is active
	drive.Config.params[2].datalen := 4;

	//Motor Data
	drive.Config.params[3].index := 16#4063;	//Motor Nominal Voltage 99.07
	drive.Config.params[3].subIndex := 16#7;
	drive.Config.params[3].data := 4150;	//415V
	drive.Config.params[3].datalen := 4;

	drive.Config.params[4].index := 16#4063;	//Motor Nominal Frequency 99.08
	drive.Config.params[4].subIndex := 16#8;
	drive.Config.params[4].data := 5000;	//50Hz
	drive.Config.params[4].datalen := 4;

	drive.Config.params[5].index := 16#4063;	//Motor Power Factor 99.11
	drive.Config.params[5].subIndex := 16#B;
	drive.Config.params[5].data := 80;	//0.8
	drive.Config.params[5].datalen := 4;

	drive.Config.params[6].index := 16#4063;	//Motor Control Mode 99.04
	drive.Config.params[6].subIndex := 16#4;
	drive.Config.params[6].data := 1;	//Scalor
	drive.Config.params[6].datalen := 2;

	//Limits
	drive.Config.params[7].index := 16#401E;	//Max Current 30.17
	drive.Config.params[7].subIndex := 16#11;
	drive.Config.params[7].data := maxCurrent;
	drive.Config.params[7].datalen := 4;

	drive.Config.params[8].index := 16#401E;	//Max Frequency 30.14
	drive.Config.params[8].subIndex := 16#E;
	drive.Config.params[8].data := ABB_MAX_VELOCITY * 100;	//60Hz
	drive.Config.params[8].datalen := 4;

	//Fault Functions
	//	drive.Config.params[9].index := 16#401F;	//External Event 1 Source 31.01
	//	drive.Config.params[9].subIndex := 16#1;
	//	drive.Config.params[9].data := 2;	//Digital Input 1 Triggers Fault When Low
	//	drive.Config.params[9].datalen := 4;

	drive.Config.params[9].index := 16#4032;	//Comms loss function 50.02
	drive.Config.params[9].subIndex := 16#2;
	drive.Config.params[9].data := 1;	//Fault on comms loss
	drive.Config.params[9].datalen := 2;

	//Other
	drive.Config.params[10].index := 16#4014;	//External Commands 20.01
	drive.Config.params[10].subIndex := 16#1;
	drive.Config.params[10].data := 12;	//Fieldbus A Selected
	drive.Config.params[10].datalen := 2;

	drive.Config.params[11].index := 16#401C;	//Frequency Ext 1 Ref 28.11
	drive.Config.params[11].subIndex := 16#B;
	drive.Config.params[11].data := 4;	//Fieldbus A As Ref
	drive.Config.params[11].datalen := 4;

	drive.Config.params[12].index := 16#401F;	//STO Indication 31.22
	drive.Config.params[12].subIndex := 16#16;
	drive.Config.params[12].data := 3;	//Warning/Warning
	drive.Config.params[12].datalen := 2;

	drive.Config.params[13].index := 16#4013;	//Disable local mode 19.17
	drive.Config.params[13].subIndex := 16#11;
	drive.Config.params[13].data := BOOL_TO_DINT(NOT Std.Drives_AllowLocalMode);// 0 = Enabled ,1 = Locked
	drive.Config.params[13].datalen := 2;

	drive.Config.params[14].index := 16#4032;	//Comm loss time out 50.03
	drive.Config.params[14].subIndex := 16#3;
	drive.Config.params[14].data := 15;	//1 second
	drive.Config.params[14].datalen := 2;

	drive.Config.params[15].index := 16#401E;	//Min Frequency 30.13
	drive.Config.params[15].subIndex := 16#D;
	drive.Config.params[15].data := ABB_MAX_VELOCITY * -100;
	drive.Config.params[15].datalen := 4;

	drive.Config.params[16].index := 16#4063;	//Nominal Current 9906
	drive.Config.params[16].subIndex := 16#6;
	drive.Config.params[16].data := nominalCurrent_9906;
	drive.Config.params[16].datalen := 4;

	drive.Config.params[17].index := 16#4063;	//Nominal Speed 9909
	drive.Config.params[17].subIndex := 16#9;
	drive.Config.params[17].data := nominalSpeed_9909;
	drive.Config.params[17].datalen := 4;

	drive.Config.params[18].index := 16#4063;	//Nominal Power 9910
	drive.Config.params[18].subIndex := 16#A;
	drive.Config.params[18].data := nominalPower_9910;
	drive.Config.params[18].datalen := 4;

	drive.Config.params[19].index := 16#401C;	//Acc time 2872  1500 = 1.5secs
	drive.Config.params[19].subIndex := 16#48;
	drive.Config.params[19].data := accTime;
	drive.Config.params[19].datalen := 4;

	drive.Config.params[20].index := 16#401C;	//Dec time 2873
	drive.Config.params[20].subIndex := 16#49;
	drive.Config.params[20].data := decTime;
	drive.Config.params[20].datalen := 4;

END_ACTION
```

#### setParameters.st
```iecst
ACTION _setParameters:

	CASE settings.MotorSize OF // Need to set these values correctly

		ABB_MOTOR_0_25KW:
			nominalCurrent_9906		:= 7; //0.68 A
			nominalPower_9910		:= 25; // 0.37 kW
			nominalSpeed_9909 		:= 1300;
			maxCurrent				:= 190;//1.9A

		ABB_MOTOR_0_37KW_0_91A_1374:
			nominalCurrent_9906		:= 9; //0.91 A
			nominalPower_9910		:= 37; // 0.37 kW
			nominalSpeed_9909 		:= 1374;
			maxCurrent 				:= 320; //3.2A

		ABB_MOTOR_0_37KW_0_97A_1342:
			nominalCurrent_9906		:= 10; //0.97 A
			nominalPower_9910		:= 37; // 0.37 kW
			nominalSpeed_9909 		:= 1342;
			maxCurrent 				:= 350; //3.5A

		ABB_MOTOR_0_37KW_1_14A_1380:
			nominalCurrent_9906		:= 7; //1.14 A
			nominalPower_9910		:= 37; // 0.37 kW
			nominalSpeed_9909 		:= 1380;
			maxCurrent 				:= 350;//3.5A

		ABB_MOTOR_0_75KW:
			nominalCurrent_9906		:= 18; //1.75 A
			nominalPower_9910		:= 75; // 0.75 kW
			nominalSpeed_9909 		:= 1440;
			maxCurrent 				:= 1170; //11.7A

		ABB_MOTOR_1_5KW:
			nominalCurrent_9906		:= 30;// 3 A?
			nominalPower_9910		:= 150;// 1.5kW
			nominalSpeed_9909 		:= 1450;
			maxCurrent 				:= 2200; //22A ???

		ABB_MOTOR_2_2KW_4_75A_1450:
			nominalCurrent_9906		:= 48; //4.75 A
			nominalPower_9910		:= 220; // 2.2 kW
			nominalSpeed_9909 		:= 1450;
			maxCurrent 				:= 3000; //30A ???

		ABB_MOTOR_3KW:
			nominalCurrent_9906		:= 64;
			nominalPower_9910		:= 300; // 3 kW
			nominalSpeed_9909 		:= 1456;
			maxCurrent 				:= 5248; //52.48

		ABB_MOTOR_CUSTOM: // Future  Alow Motor data to be set individaully
			nominalCurrent_9906		:= 26; //2.55A
			nominalPower_9910		:= 110; //1.1
			nominalSpeed_9909 		:= 1455;
			maxCurrent 				:= 1760; //17.6A

	END_CASE;

	accTime := REAL_TO_DINT(settings.AccTime * 1000);
	decTime := REAL_TO_DINT(settings.DecTime * 1000);

	//V2.00.2 Encode parameters
	_encodeParameters;

	drive.Config.function.enable := TRUE;																	//Enable function block

	IF (drive.Config.Node > 0) THEN
		drive.Config.function.node := drive.Config.Node; 														//Node number of drive, set in ABB_EPL[n].cmd.node if non standard.
		drive.Config.function.pDevice := ADR(drive.Config.EPL_Address);											//Set powerlink address in ABB_Driver init task
	ELSE
		//drive.Config.function.node := n + 100; //Set the default to drive + 100
	END_IF;
	IF (drive.Config.Node > 0) AND (drive.Config.currentParam <= MAX_PARAMS) THEN
		IF (drive.Config.params[drive.Config.currentParam].status > 0) THEN									//Call function only if not completed
			drive.Config.function.index := drive.Config.params[drive.Config.currentParam].index; 			//Powerlink index address
			drive.Config.function.subindex := drive.Config.params[drive.Config.currentParam].subIndex;		//Powerlink sub index address
			drive.Config.function.pData := ADR(drive.Config.params[drive.Config.currentParam].data);		//Value of data to write
			drive.Config.function.datalen := drive.Config.params[drive.Config.currentParam].datalen;		//Size of data type														//Call function
			IF (drive.Config.function.status = ERR_OK) THEN 												//Clear errors
				drive.Config.params[drive.Config.currentParam].status := 0;
				drive.Config.params[drive.Config.currentParam].errorInfo := 0;
				drive.Config.currentParam := drive.Config.currentParam + 1;
			ELSIF (drive.Config.function.status <> ERR_FUB_BUSY) AND (drive.Config.function.status <> ERR_FUB_ENABLE_FALSE) THEN //Store errors
				drive.Config.params[drive.Config.currentParam].status := drive.Config.function.status;
				drive.Config.params[drive.Config.currentParam].errorInfo := drive.Config.function.errorinfo;
				drive.Config.function.enable := FALSE;
				//			ELSIF drive.Config.function.status <> 20925 THEN;//ERR_PLMGR_STATION_NOT_ACTIVE THEN  //Only skip if the devuce is active																																					//Skip if other error to stop PLC hanging in bootup
				//				drive.Config.params[drive.Config.currentParam].status := drive.Config.function.status;
				//				drive.Config.params[drive.Config.currentParam].errorInfo := drive.Config.function.errorinfo;
				//				drive.Config.currentParam := drive.Config.currentParam + 1;
			END_IF;
			drive.Config.function();
		ELSE
			drive.Config.function.enable := FALSE;
		END_IF;
	END_IF;

	//Parameters should be loaded onto default settings.
	//to default the drive set 9606 t0 34560
	//Node ID (5103) has to be manually set

END_ACTION
```

#### _manual.st
```iecst
//Manual Mode
ACTION _manual:

	//visu_drive is an array which contains the array index of the drive we want to see.

	FOR n := 1 TO max_manualControls DO

		visu_man ACCESS ADR(visu_manual[n]);

		selIndex := atoi(ADR(visu_man.selectedValue));
		IF (selIndex > 0) AND (selIndex <= MAX_DRIVES) AND (selIndex <> visu_man.selectedIndex) THEN
			updateDropDown := 1;
			visu_man.selectedIndex := DINT_TO_UINT(selIndex);
		END_IF;

		visu_man.ListBoxVisible := (visu_man.selectedIndex = 0);

		visu_man.refreshDropDown.CLK := (visu_man.selectedIndex = 0);
		visu_man.refreshDropDown();
		IF visu_man.refreshDropDown.Q THEN
			updateDropDown := 1;
		END_IF;

		drive ACCESS ADR(ABB_EPL.Drives[visu_man.selectedIndex]);
		drive.Manual.Enable 	:= 1; // Mark the drive as in manual mode.
		drive.Manual.Velocity 	:= visu_man.TargetVelocity;

		visu_man.Visible		:= (visu_man.selectedIndex > 0);
		visu_man.Name			:= gSettings.Drive[visu_man.selectedIndex].Name;
		visu_man.Node		 	:= drive.Config.Node;
		visu_man.ModuleOk 		:= drive.Comm.ModuleOk;
		visu_man.ActVelocity 	:= ABS(drive.Comm.ActVelocity);
		visu_man.ActCurrent 	:= drive.Comm.ActCurrent;
		visu_man.ActTorque 		:= drive.Comm.ActTorque;
		visu_man.ErrorCode 		:= drive.Comm.ErrorCode;

		visu_man.ErrorActive	:= (drive.Comm.State = ABB_TRIPPED);

		IF visu_man.ErrorReset THEN
			visu_man.ErrorReset := 0;
			drive.Manual.ErrorReset := 1;
		END_IF;

		CASE drive.Comm.State OF
			ABB_INIT:
				visu_man.State := '$$Drives.State.Init';
			ABB_DISCONNECTED:
				visu_man.State := '$$Drives.State.Disconnected';
			ABB_QUICK_STOP:
				visu_man.State := '$$Drives.State.QuickStop';
			ABB_CONFIG:
				visu_man.State := '$$Drives.State.Config';
			ABB_SWITCH_ON_INHIBITED:
				visu_man.State := '$$Drives.State.SwitchOnInhibit';
			ABB_NOT_READY_TO_SWITCH_ON:
				visu_man.State := '$$Drives.State.NotReady';
			ABB_READY_TO_SWITCH_ON:
				visu_man.State := '$$Drives.State.ReadyToSwitchOn';
			ABB_READY_TO_RUN:
				visu_man.State := '$$Drives.State.ReadyToRun';
			ABB_RUNNING:
				visu_man.State := '$$Drives.State.Running';
			ABB_TRIPPED:
				visu_man.State := '$$Drives.State.Tripped';
			ABB_OFF_REMOTE:
				visu_man.State := '$$Drives.State.OffRemote';
			ABB_STO:
				visu_man.State := '$$Drives.State.STO';
			ABB_RAMP_DOWN:
				visu_man.State := '$$Drives.State.RampDown';
			ELSE
				visu_man.State := '';
		END_CASE;

		targetSpeedValid := ((visu_man.TargetVelocity >= ABB_MIN_VELOCITY) AND (visu_man.TargetVelocity <= ABB_MAX_VELOCITY) AND ((drive.Comm.State = ABB_READY_TO_RUN) OR  (drive.Comm.State = ABB_RUNNING)));

		IF NOT targetSpeedValid THEN
			visu_man.RunReverse 		:= 0;
			visu_man.RunForwards 		:= 0;
			visu_man.EnableRunReverse 	:= 0;
			visu_man.EnableRunForwards 	:= 0;
		ELSIF visu_man.RunForwards THEN
			drive.Manual.Direction 	:= ABB_DIRECTION_FWD;
			drive.Manual.Run		:= targetSpeedValid;
			visu_man.EnableRunReverse := 0;
		ELSIF visu_man.RunReverse THEN
			drive.Manual.Direction 	:= ABB_DIRECTION_REV;
			drive.Manual.Run		:= targetSpeedValid;
			visu_man.EnableRunForwards := 0;
		ELSE
			visu_man.EnableRunReverse := 1;
			visu_man.EnableRunForwards := 1;
			drive.Manual.Run		:= 0;
		END_IF;

	END_FOR;

	//Build the list box string;
	//[{'value':'text_1', 'text':'$$IAT/testText1'}, {'value':'text_2', 'text':'$$IAT/testText2'}]
	IF updateDropDown THEN
		index := 1;
		brsmemset(ADR(manualSelectDrowDown),0,SIZEOF(manualSelectDrowDown));
		manualSelectDrowDown[0] := '{"value":0,"text":""}';
		FOR n := 1 TO MAX_DRIVES DO
			drive ACCESS ADR(ABB_EPL.Drives[n]);
			IF NOT drive.Manual.Enable THEN
				itoa(n,ADR(sIndex));
				brsstrcat(ADR(manualSelectDrowDown[index]),ADR('{"value":"'));
				brsstrcat(ADR(manualSelectDrowDown[index]),ADR(sIndex));
				brsstrcat(ADR(manualSelectDrowDown[index]),ADR('","text":"'));
				brsstrcat(ADR(manualSelectDrowDown[index]),ADR(gSettings.Drive[n].Name));
				brsstrcat(ADR(manualSelectDrowDown[index]),ADR('"}'));
				index := index + 1;
			END_IF;
		END_FOR;
		updateDropDown := FALSE;
	END_IF;

END_ACTION
```

#### _getNodeInfo.st
```iecst
ACTION _getNodeInfo:
	IF (index >= 1) AND (index <= MAX_DRIVES) THEN//  AND (LEN(POWERLINK_INTERFACE_ADDRESS) > 0) THEN
		config ACCESS ADR (ABB_EPL.Drives[index].Config);

		CASE init_state OF
			0:
				IF (config.Node = 0) THEN
					pvName := 'ABB_EPL.Drives[';
					itoa(index,ADR(driveNo));
					brsstrcat(ADR(pvName),ADR(driveNo));
					brsstrcat(ADR(pvName),ADR(']'));
					getNode.enable := 1;
					getNode.pvName := pvName;
					getNode();
					IF (getNode.status = ERR_OK) THEN
						config.Node 		:= getNode.NodeNumber;
						config.EPL_Address 	:= getNode.IF_Adr;
						// Build the path for the name
						itoa(getNode.NodeNumber,ADR(sNode));
						moduleAddress := CONCAT(getNode.IF_Adr,'.ST');
						moduleAddress := CONCAT(moduleAddress,sNode);
						init_state := 1;
					ELSIF (getNode.status <> ERR_FUB_BUSY) THEN
						init_state := 10; // SKIP -- CAMERA HASN'T BEEN MAPPED
					END_IF;
				ELSE
					init_state := 10; // SKIP -- CAMERA HASN'T BEEN MAPPED
				END_IF

			1: //Get the name if it hasn;t be set
				IF (gSettings.Drive[index].Name = '') THEN
					getModuleName.enable := 1;
					getModuleName.pModuleAddress := ADR(moduleAddress);
					getModuleName();
					IF getModuleName.status = ERR_OK THEN
						init_state := 10;
						gSettings.Drive[index].Name := LEFT(getModuleName.ModuleName,SIZEOF(gSettings.Drive[index].Name));
					ELSIF (getModuleName.status <> ERR_FUB_BUSY) THEN
						gSettings.Drive[index].Name := 'unknown';
						init_state := 10;
					END_IF;
				ELSE
					init_state := 10;
				END_IF;

			10:// Done
				index := index + 1;
				init_state := 0;
			ELSE
				index := index + 1;
				init_state := 0;
		END_CASE;

	ELSIF (index < 1) THEN
		index := 1;
	ELSIF index > MAX_DRIVES THEN
		xRun := 1;
	END_IF;

END_ACTION
```

#### _packData.st
```iecst
ACTION _packData:

	IF drive.Cmd.Run THEN
		CASE drive.Cmd.Direction OF

			ABB_DIRECTION_FWD:
				drive.Comm.TargetVelocity :=	drive.Cmd.TargetVelocity;

			ABB_DIRECTION_REV:
				drive.Comm.TargetVelocity :=	drive.Cmd.TargetVelocity * - 1;
		END_CASE;
	ELSIF drive.Manual.Run THEN
		CASE drive.Manual.Direction OF

			ABB_DIRECTION_FWD:
				drive.Comm.TargetVelocity :=	drive.Manual.Velocity;
			ABB_DIRECTION_REV:
				drive.Comm.TargetVelocity :=	drive.Manual.Velocity * - 1;
			ELSE
				drive.Comm.TargetVelocity :=	drive.Manual.Velocity;
		END_CASE;
	END_IF;

	//Control Word																Status Word
	//Bit 0		Switch On														Bit 0		Ready To Switch On
	//Bit 1		Enable Voltage											Bit 1		Switched On
	//Bit 2		Quick Stop													Bit 2		Operation Enabled
	//Bit 3		Enable Operation										Bit 3		Fault
	//Bit 4		Not Used In Scalor Mode							Bit 4		Voltage Enabled
	//Bit 5		Not Used In Scalor Mode							Bit 5		Quick Stop
	//Bit 6		Not Used In Scalor Mode							Bit 6		Switch On Disabled
	//Bit 7		Fault Reset													Bit 7 	Warning
	//Bit 8		Halt																Bit 8		Drive Specific TBC
	//Bit 9		Operation Mode Specific							Bit 9		Remote
	//Bit 10	Reserved	??Remote Control??				Bit 10	Target Reached
	//Bit 11	Drive Specific	TBC									Bit 11 	Internal Limit Reached
	//Bit 12	Drive Specific	TBC									Bit 12	Not Used In Scalor Mode
	//Bit 13	Drive Specific	TBC									Bit 13	Not Used In Scalor Mode
	//Bit 14	Drive Specific	TBC									Bit 14	Drive Specific TBC
	//Bit 15	Drive Specific	TBC									Bit 15	Drive Specific TBC

	drive.Status.ReadyToSwitchOn 	:= drive.Comm.StatusWord.0;
	drive.Status.ReadyToRun 		:= drive.Comm.StatusWord.1;
	drive.Comm.StatusWord.2; //Ready to ref-- not used
	drive.Status.Tripped 			:= drive.Comm.StatusWord.3;
	drive.Status.DriveEnabled 	:= drive.Comm.StatusWord.4; //the drive is enabled..
	drive.Status.QuickstopActive 	:= NOT drive.Comm.StatusWord.5; //QuickStop is not active
	drive.Status.SwitchOnInhibit 	:= drive.Comm.StatusWord.6; //We can't enable the drive....
	drive.Status.Warning 			:= drive.Comm.StatusWord.7;
	drive.Status.AtSpeed 			:= drive.Comm.StatusWord.8;
	drive.Status.OnRemote 		:= drive.Comm.StatusWord.9;

	drive.Status.ActCurrent := drive.Comm.ActCurrent;
	drive.Status.ActTorque := drive.Comm.ActTorque;

	//drive.Status.ThermalTrip := drive.Comm.DI.0;

END_ACTION
```

- ABB Drive Commissioning Guide.docx - Commissioning guide (binary file, 20887 bytes)
### Program Logical/Standard/Barcode_BnR/Camera_Driver (IEC, version 1.00.6) - *Needs 10ms  Controller task for all BnR Barcode readers. and MappView Handling

#### Main.st - Init, cyclic, exit code
```iecst
//V1.00.1 TR. 15/12/2020: ADD: Automatically populate camera ip and node.
//V1.00.2 TR. 19/02/2021: ADD: Allow auto tune when the image is not ready, Init focus/exposure settings.
//V1.00.3 TR  22/02/2021: ADD: New pre check state. to allow the camera to load its firmware without setting any bits.
//V1.00.4 TR  22/02/2021: UPDATE: Update to match new mappview -- Change the image widget from web view to image..
//V1.00.5 TR 	26/05/2021: FIX: Camera could get stuck on the GET_IMAGE_STEP -> Added a retry timeout.
//V1.00.6 TR 	19/10/2021: ADD: Explicit state for retrying on time out, so we are sure to generate an edge on the Read command.

//http://10.8.4.20:81/index.html?visuid=mappvision  < -- DO NOT USE THIS ITS POOP

//?? Should we make auto retune on failure an option. or should the requester handle this on read fail?
//We can use the asHW TO detect when the camera is plugged into the system OR NOT as automatically make it visibile?

PROGRAM _INIT
	lastID 	:= 0;
	index 	:= 1;

	FOR n := 1 TO MAX_CAMERAS DO
		camera 		ACCESS ADR(Camera[n]);
		settings 	ACCESS ADR(gSettings.Camera[n]);
		camera.Internal.state := CAMERA_LOAD_SETTINGS;
		//Initialise the fixed settings.
		settings.FlashColour 	:= 1;
		settings.FlashSegment 	:= 15;
		settings.NumSearchMax 	:= 1;
		settings.SymbolType 	:= 50;
		settings.Timeout		:= 50; // If set to 0 this is handled by the camera.

		IF (settings.Focus = 0) THEN settings.Focus := 1700; END_IF;
		IF (settings.Exposure = 0) THEN settings.Exposure := 35; END_IF;

		IF (settings.ReadCount = 0) THEN settings.ReadCount := 5; END_IF;
	END_FOR;

	xRun 	:= FALSE;
	init 	:= 0;
	index 	:= 0;
END_PROGRAM

PROGRAM _CYCLIC

	IF EDGENEG(xRun) THEN
		FOR n := 1 TO MAX_CAMERAS DO
			Camera[n].Node := 0;
		END_FOR;
		index 	:= 0;
		init 	:= 0;
	ELSIF NOT xRun THEN
		_initPaths;
	ELSE
		FOR n := 1 TO MAX_CAMERAS DO
			camera 		ACCESS ADR(Camera[n]);
			settings 	ACCESS ADR(gSettings.Camera[n]);
			state 		ACCESS ADR(camera.Internal.state);

			camera.Errors.OS_check := camera.Info.Status.24;
			camera.Errors.VA_loading := camera.Info.Status.25;

			IF camera.Errors.OS_check OR camera.Errors.VA_loading THEN
				state := CAMERA_BOOTING;
			ELSIF camera.Errors.UnderVoltage THEN
				state := CAMERA_ERROR;
			ELSIF NOT camera.ModuleOk THEN
				state := CAMERA_NOT_PRESENT;
			END_IF;

			CASE state OF
				CAMERA_LOAD_SETTINGS: // Load the settings from the camera setting area
					camera.Parameters.Write.Focus 			:= settings.Focus;
					camera.Parameters.Write.Gain 			:= settings.Gain;
					camera.Parameters.Write.Exposure 		:= settings.Exposure;
					camera.Parameters.Write.FlashSegment 	:= settings.FlashSegment;
					camera.Parameters.Write.FlashColour 	:= settings.FlashColour;
					camera.Parameters.Write.NumSearchMax 	:= settings.NumSearchMax;
					camera.Parameters.Write.SymbolType	 	:= settings.SymbolType;
					camera.Parameters.Write.Timeout	 		:= settings.Timeout;
					camera.Internal.readCount				:= 0;
					IF camera.Info.ImageAcquisitionReady THEN
						state := CAMERA_READY;
					ELSE
						state := CAMERA_NOT_READY;
					END_IF;

				CAMERA_READY:
					IF NOT camera.Info.ImageAcquisitionReady THEN
						state := CAMERA_NOT_READY;
					ELSIF camera.Interface.Read OR visu.cmd.Capture THEN
						state := CAMERA_GET_IMAGE;
					ELSIF camera.Interface.AutoTune OR visu.cmd.AutoTune THEN
						state := CAMERA_AUTO_TEACH;
					END_IF;

				CAMERA_GET_IMAGE:
					IF camera.Functions.ImageAquisitionComplete.Q THEN
						camera.Internal.readCount := camera.Internal.readCount + 1;
						IF (camera.Info.NumResults > 0) THEN
							brsstrcpy(ADR(camera.Interface.Result),ADR(camera.Results));
							state := CAMERA_RESULT_ACQUIRED;
						ELSE
							state := CAMERA_RESET;
						END_IF;
					ELSIF camera.Functions.TonRetry.Q THEN
						state := CAMERA_RESET;
					END_IF;

				CAMERA_RESULT_ACQUIRED:
					IF NOT camera.Interface.Read AND NOT visu.cmd.Capture THEN
						IF NOT camera.Info.ImageAcquisitionReady THEN
							state := CAMERA_NOT_READY;
						ELSE
							state := CAMERA_RESET;
						END_IF;
					END_IF;

				CAMERA_AUTO_TEACH:
					IF camera.Info.Status > 0 THEN
						camera.Internal.tuning := 1;
					END_IF;
					IF camera.Functions.AutoTuneComplete.Q THEN
						settings.Exposure := camera.Parameters.Read.Exposure;
						settings.Focus := camera.Parameters.Read.Focus;
						settings.Gain := camera.Parameters.Read.Gain;
						state := CAMERA_AUTO_TEACH_DONE;
					END_IF;

				CAMERA_AUTO_TEACH_DONE:
					IF NOT camera.Interface.AutoTune AND NOT visu.cmd.AutoTune THEN
						state := CAMERA_LOAD_SETTINGS;
					END_IF;

				CAMERA_NOT_READY:
					IF camera.Info.ImageAcquisitionReady THEN
						state := CAMERA_LOAD_SETTINGS;
					ELSIF camera.Interface.AutoTune OR visu.cmd.AutoTune THEN
						state := CAMERA_AUTO_TEACH;
					END_IF;

				CAMERA_BOOTING: //loading OS or updating firmare.
					IF NOT camera.Errors.OS_check AND NOT camera.Errors.VA_loading THEN
						state := CAMERA_LOAD_SETTINGS;
					END_IF;

				CAMERA_RESET:
					IF camera.Functions.TonReset.Q THEN
						state := CAMERA_READY;
					END_IF;

				CAMERA_NOT_PRESENT:
					IF camera.ModuleOk THEN
						state := CAMERA_LOAD_SETTINGS;
					END_IF;

				CAMERA_ERROR:
					IF NOT camera.Errors.UnderVoltage THEN
						state := CAMERA_LOAD_SETTINGS;
					END_IF;

			END_CASE;

			camera.Parameters.Write.Read := (state = CAMERA_GET_IMAGE);
			camera.Interface.ResultReady := (state = CAMERA_RESULT_ACQUIRED);
			camera.Parameters.Write.Enable := ((state = CAMERA_READY) OR (state = CAMERA_RESULT_ACQUIRED) OR (state = CAMERA_GET_IMAGE));
			camera.Parameters.Write.SearchAcquisitionSettings := (state = CAMERA_AUTO_TEACH);

			camera.Functions.TonRetry.IN := (state = CAMERA_GET_IMAGE) AND NOT camera.Info.ImageProcessingActive;
			camera.Functions.TonRetry.PT := T#2s;
			camera.Functions.TonRetry();

			camera.Functions.TonReset.IN := (state = CAMERA_RESET);
			camera.Functions.TonReset.PT := T#100ms;
			camera.Functions.TonReset();

			camera.Functions.AutoTuneComplete.CLK := (camera.Internal.tuning AND (camera.Info.Status = 0));
			camera.Functions.AutoTuneComplete();

			camera.Functions.ClearResults.CLK := (state = CAMERA_RESULT_ACQUIRED);
			camera.Functions.ClearResults();

			camera.Functions.ImageAquisitionComplete.CLK :=	camera.Info.ImageProcessingActive;
			camera.Functions.ImageAquisitionComplete();

			camera.Functions.ReadEdgeNeg.CLK := camera.Interface.Read;
			camera.Functions.ReadEdgeNeg();

			IF camera.Functions.ReadEdgeNeg.Q THEN
				camera.Internal.readCount := 0;
			END_IF;

			IF camera.Functions.ClearResults.Q THEN
				brsstrcpy(ADR(camera.Interface.Result),ADR(''));
				camera.Internal.readCount := 0;
			END_IF;

			camera.Interface.ReadFail := (camera.Internal.readCount >= settings.ReadCount);

			IF (state = CAMERA_AUTO_TEACH) THEN
				camera.Parameters.Write.StatusLED := CAMERA_LED_BLUE;
			ELSIF (state = CAMERA_AUTO_TEACH_DONE) THEN
				IF Std.Clock1s THEN
					camera.Parameters.Write.StatusLED := CAMERA_LED_BLUE;
				ELSE
					camera.Parameters.Write.StatusLED := CAMERA_LED_DISABLED;
				END_IF;
			ELSIF camera.Interface.ReadFail THEN
				camera.Parameters.Write.StatusLED := CAMERA_LED_RED;
			ELSE
				camera.Parameters.Write.StatusLED := CAMERA_LED_AUTO;
			END_IF;

			IF (state <> CAMERA_AUTO_TEACH) THEN
				camera.Internal.tuning := 0;
			END_IF;

			camera.Interface.Ready := (state = CAMERA_READY) AND (NOT visu.cmd.Repeat OR (visu.cameraID <> n));
			camera.Parameters.Write.ResetAcquisitionSettings := (state = CAMERA_NOT_READY);
			camera.Interface.AutoTuneDone := (state = CAMERA_AUTO_TEACH_DONE);

		END_FOR;

		//Control for MappView

		_visuControl;

	END_IF;

END_PROGRAM

PROGRAM _EXIT
	(* Insert code here *)

END_PROGRAM
```

#### _initPaths.st
```iecst
//Build the WEB URL for the camera images..
//Only do it once..
ACTION _initPaths:

	IF (index >= 1) AND (index <= MAX_CAMERAS) THEN//  AND (LEN(POWERLINK_INTERFACE_ADDRESS) > 0) THEN
		CASE init OF
			0: // Get the Node number

				pvName := 'Camera[';
				itoa(index,ADR(camNo));
				brsstrcat(ADR(pvName),ADR(camNo));
				brsstrcat(ADR(pvName),ADR(']'));
				getNode.enable := 1;
				getNode.pvName := pvName;
				getNode();
				IF (getNode.status = ERR_OK) THEN
					Camera[index].Node := getNode.NodeNumber;
					itoa(getNode.NodeNumber,ADR(sNode));
					init := 1;
				ELSIF (getNode.status <> ERR_FUB_BUSY) THEN
					init := 10;	 // SKIP -- CAMERA HASN'T BEEN MAPPED
				END_IF;

			1:
				getPowerlinkNodeIP();
				//Initialise the Camera values for Visu
				getPowerlinkNodeIP.EplInterfacePath 	:= getNode.IF_Adr;//POWERLINK_INTERFACE_ADDRESS;
				getPowerlinkNodeIP.pIPAddress			:= ADR(eplIpAddress);
				getPowerlinkNodeIP.Enable := 1;
				getPowerlinkNodeIP.Node 	:= USINT_TO_UDINT(Camera[index].Node);

				IF (getPowerlinkNodeIP.Status = ERR_OK) THEN
					//Build the URL
					web_path[index]	:= 'http://';
					web_path[index] := CONCAT(web_path[index],eplIpAddress);
					web_path[index]:= CONCAT(web_path[index],':8080/jpg?q=50,t=');
					getPowerlinkNodeIP.Enable := 0;
					init := 2;
				ELSIF (getPowerlinkNodeIP.Status <> ERR_FUB_BUSY) AND (getPowerlinkNodeIP.Status <> ERR_FUB_ENABLE_FALSE) THEN
					web_path[index]	:= '';
					init := 2;
					getPowerlinkNodeIP.Enable := 0;
				END_IF;

			2:// Get the camera name
				IF (gSettings.Camera[index].Name = '') THEN
					moduleAddress := CONCAT(getNode.IF_Adr,'.ST');
					moduleAddress := CONCAT(moduleAddress,sNode);

					getModuleName.enable := 1;
					getModuleName.pModuleAddress := ADR(moduleAddress);
					getModuleName();
					IF getModuleName.status = ERR_OK THEN
						init := 10;
						gSettings.Camera[index].Name := LEFT(getModuleName.ModuleName,SIZEOF(gSettings.Camera[index].Name));
					ELSIF (getModuleName.status <> ERR_FUB_BUSY) THEN
						gSettings.Camera[index].Name := 'unknown';
						init := 10;
					END_IF;
				ELSE
					init := 10;
				END_IF;

			10://
				init := 0;
				index := index + 1;

		END_CASE;

	ELSIF (index < 1) THEN
		index := 1;
	ELSIF index > MAX_CAMERAS THEN
		xRun := 1;
	END_IF;

END_ACTION
```

#### _visuControl.st
```iecst
//Visualisation controll
ACTION _visuControl:

	//Set the index of the camera we are looking at.
	IF (visu.cameraID <= 0) THEN
		visu.cameraID := MAX_CAMERAS;
	ELSIF (visu.cameraID > MAX_CAMERAS) THEN
		visu.cameraID := 1;
	END_IF;

	visu_camera 	ACCESS ADR(Camera[visu.cameraID]);
	visu_settings 	ACCESS ADR(gSettings.Camera[visu.cameraID]);
	state 			ACCESS ADR(visu_camera.Internal.state);

	IF (visu.cameraID <> lastID) THEN

		visu.reload 		:= 1;
		lastID 				:= visu.cameraID;
	END_IF;

	IF EDGEPOS(visu.cmd.AutoTune AND state = CAMERA_AUTO_TEACH_DONE) THEN
		visu.cmd.AutoTune := 0;
	END_IF;

	IF visu_camera.Functions.ImageAquisitionComplete.Q AND visu.cmd.Capture  THEN
		visu.reload 		:= 1;
		visu.cmd.Capture 	:= 0;
		visu_camera.Internal.readCount := 0; //Reset the read count as the image was manually triggered
	END_IF;

	tof_repeat.IN := (visu_camera.Functions.ImageAquisitionComplete.Q AND visu.cmd.Repeat);
	tof_repeat.PT := T#250ms;//4FPS
	tof_repeat();

	IF EDGENEG(tof_repeat.Q) THEN
		visu.cmd.Capture := 1;
	END_IF;

	IF EDGEPOS( visu.cmd.Repeat) THEN
		IF (state = CAMERA_READY) THEN
			visu.cmd.Capture := 1;
		ELSE
			visu.cmd.Repeat := 0;
		END_IF;
	END_IF;

	IF visu.reload THEN // Build a path with the timestamp so we can force the mapp image widget to update.
		//'http://192.168.201.17:8080/jpg?q=50t={timevalue}';
		itoa(ABS(clock_ms()),ADR(timeString));
		buildURL := web_path[visu.cameraID];
		brsstrcat(ADR(buildURL),ADR(timeString));
		visu.ImageAddress := buildURL;
		visu.reload := 0;
	END_IF;

	IF EDGEPOS(visu.cmd.SaveSettings) THEN
		camera.Parameters.Write.Focus 			:= settings.Focus;
		camera.Parameters.Write.Gain 			:= settings.Gain;
		camera.Parameters.Write.Exposure 		:= settings.Exposure;
		//		camera.Parameters.Write.FlashSegment 	:= settings.FlashSegment;
		//		camera.Parameters.Write.FlashColour 	:= settings.FlashColour;
		//		camera.Parameters.Write.NumSearchMax 	:= settings.NumSearchMax;
		//		camera.Parameters.Write.SymbolType	 	:= settings.SymbolType;
		camera.Parameters.Write.Timeout	 		:= settings.Timeout;
		visu.cmd.SaveSettings := 0;
	END_IF;

	visu.voltageOk := visu_camera.ModuleOk AND NOT visu_camera.Errors.UnderVoltage;

	visu.buttonEnable.Tune 		:= (((state = CAMERA_READY) OR (state = CAMERA_AUTO_TEACH_DONE) OR (state = CAMERA_NOT_READY)) AND NOT visu.cmd.Repeat);
	visu.buttonEnable.Capture 	:= ((state = CAMERA_READY) OR visu.cmd.Capture) AND NOT visu.cmd.Repeat;
	visu.buttonEnable.Repeat 	:= ((state = CAMERA_READY) OR visu.cmd.Repeat);
	visu.enableSettings			:= (state <> CAMERA_AUTO_TEACH);

END_ACTION
```

#### Types.typ - Local data types
```iecst
TYPE
	visu_typ : 	STRUCT  (**Data type for camera mappview*)
		cameraID : USINT; (**ID of the camera we are looking at.*)
		reload : BOOL; (**Command to reload the web viewer*)
		cmd : visu_cmd_typ;
		voltageOk : BOOL;
		ImageAddress : STRING[100]; (**Ip Address of Image Path*)
		buttonEnable : visu_btn_status_typ;
		enableSettings : BOOL; (**Enable input of manually setting camera settings.*)
	END_STRUCT;
	visu_cmd_typ : 	STRUCT
		AutoTune : BOOL; (**Auto Tune*)
		Capture : BOOL; (**Get a single image*)
		Repeat : BOOL; (**Repeat capture image*)
		SaveSettings : BOOL; (**Apply the setting values*)
	END_STRUCT;
	visu_btn_status_typ : 	STRUCT
		Tune : BOOL;
		Repeat : BOOL;
		Capture : BOOL;
	END_STRUCT;
END_TYPE
```

#### Variables.var - Local variables
```iecst
VAR
	visu : visu_typ;
	n : USINT;
	visu_camera : REFERENCE TO Camera_typ;
	camera : REFERENCE TO Camera_typ;
	state : REFERENCE TO Camera_state_enum;
	settings : REFERENCE TO Camera_Settings_typ;
	tof_repeat : TOF;
	visu_settings : REFERENCE TO Camera_Settings_typ;
	lastID : USINT;
	getPowerlinkNodeIP : GetPowerlinkNodeIP;
	eplIpAddress : STRING[16];
	web_path : ARRAY[0..MAX_CAMERAS] OF STRING[50];
	index : USINT;
	xRun : BOOL;
	getNode : getNodeFromPV;
	pvName : STRING[75];
	camNo : STRING[10];
	init : USINT;
	moduleAddress : STRING[30];
	getModuleName : GetModuleName;
	sNode : STRING[10];
	timeString : STRING[20];
	buildURL : STRING[100];
END_VAR
```

### Camera.typ
```iecst
TYPE
	Camera_typ : 	STRUCT
		ModuleOk : BOOL;
		Node : USINT; (**Node number of the camera  -- To be automatically found.*)
		Parameters : Camera_param_typ;
		Info : Camera_Info_typ;
		Results : STRING[20];
		Errors : Camera_error_typ;
		Interface : Camera_interface_typ;
		Internal : Camera_internal_typ;
		Functions : Camera_function_typ;
	END_STRUCT;
	Camera_error_typ : 	STRUCT
		UnderVoltage : BOOL;
		OS_check : BOOL; (*Operating system is loading*)
		VA_loading : BOOL; (*Visual Application is loading.*)
	END_STRUCT;
	Camera_Info_typ : 	STRUCT
		Status : UDINT;
		AcceptedAcquisitionCnt : USINT;
		CompletedAcquisitionCnt : USINT;
		FailedAcquisitionCnt : USINT;
		ImageAcquisitionReady : BOOL;
		ImageProcessingActive : BOOL;
		ImageProcessingTime : UINT;
		ImageProcessingError : UINT;
		Temperature : SINT;
		NumResults : USINT;
		FunctionProcessingTime : UINT;
	END_STRUCT;
	Camera_interface_typ : 	STRUCT
		Ready : BOOL; (**Camera is ready to read *)
		Read : BOOL; (**Set high to read the code.. Pos edge starts process. Neg Edge resets, and clears results*)
		ReadFail : BOOL; (**The read count has exceeded the maximum try count -- The camera will still try to read until the read command is removed.*)
		ResultReady : BOOL; (**Results are ready to be processed*)
		Result : STRING[20]; (**Raw string from barcode reader*)
		AutoTune : BOOL; (**Set high to autotune the camera.*)
		AutoTuneDone : BOOL; (**The camera has been successfully tuned.*)
	END_STRUCT;
	Camera_internal_typ : 	STRUCT
		state : Camera_state_enum; (**Set high to read the code.. Pos edge starts process. Neg Edge resets, and clears results*)
		readCount : UINT; (**Number of reads on each count*)
		tuning : BOOL; (**Bit when the camera is in a tuning state.*)
	END_STRUCT;
	Camera_param_read_typ : 	STRUCT
		Focus : UINT;
		Gain : USINT;
		Exposure : UDINT;
	END_STRUCT;
	Camera_param_typ : 	STRUCT
		Read : Camera_param_read_typ;
		Write : Camera_param_write_typ;
	END_STRUCT;
	Camera_param_write_typ : 	STRUCT
		Focus : UINT; (**Focus Value*)
		Gain : USINT; (**Camera Gain*)
		Exposure : UDINT; (**Camera Exposure time in uS*)
		FlashSegment : USINT; (**Sections of the Flash which should be active. 0 = All off. 15 = All on*)
		FlashColour : USINT; (**Flash color, Always 1 for RED*)
		StatusLED : USINT; (**Write to the status LED*)
		Enable : BOOL; (**Enable the barcode read function*)
		NumSearchMax : USINT; (** Number of barcodes we are looking to decode*)
		SymbolType : USINT; (**Type of barcode we are looking to decode*)
		Timeout : UINT;
		SearchAcquisitionSettings : BOOL; (**Enable Auto teach mode.*)
		ResetAcquisitionSettings : BOOL; (**Clear the results*)
		Read : BOOL; (**Command to Read*)
	END_STRUCT;
	Camera_Settings_typ : 	STRUCT
		Focus : UINT; (**Focus Value*)
		Gain : USINT; (**Camera Gain*)
		Exposure : UDINT; (**Camera Exposure time in uS*)
		FlashSegment : USINT := 15; (**Sections of the Flash which should be active. 0 = All off. 15 = All on*)
		FlashColour : USINT := 1; (**Flash color, Always 1 for RED*)
		NumSearchMax : USINT := 1; (** Number of barcodes we are looking to decode*)
		SymbolType : USINT := 50; (**Type of barcode we are looking to decode*)
		Timeout : UINT := 0;
		ReadCount : UINT := 0; (**Read count before error flag comes on*)
		Name : STRING[50]; (*'Name for idenification*)
	END_STRUCT;
	Camera_state_enum :
		(
		CAMERA_LOAD_SETTINGS := 0,
		CAMERA_READY := 1,
		CAMERA_GET_IMAGE := 2,
		CAMERA_RESULT_ACQUIRED := 3,
		CAMERA_AUTO_TEACH := 4,
		CAMERA_AUTO_TEACH_DONE := 5,
		CAMERA_NOT_READY := 6,
		CAMERA_NOT_PRESENT := 7,
		CAMERA_BOOTING := 8,
		CAMERA_RESET := 10, (**Reset between retrying to take image*)
		CAMERA_ERROR := 100
		);
	Camera_function_typ : 	STRUCT
		ClearResults : F_TRIG;
		AutoTuneComplete : R_TRIG;
		ImageAquisitionComplete : F_TRIG;
		ReadEdgeNeg : F_TRIG;
		TonRetry : TON;
		TonReset : TON;
	END_STRUCT;
END_TYPE
```

### Camera.var
```iecst
(*Constants to Set*)
(***Global Vars*)
VAR
	Camera : ARRAY[0..MAX_CAMERAS] OF Camera_typ;
END_VAR
(*Constants*)
VAR CONSTANT
	CAMERA_LED_AUTO : USINT := 0;
	CAMERA_LED_DISABLED : USINT := 1;
	CAMERA_LED_GREEN : USINT := 2;
	CAMERA_LED_RED : USINT := 3;
	CAMERA_LED_BLUE : USINT := 4;
END_VAR
```

### Standard.typ
```iecst
TYPE
	Std_Vars : 	STRUCT
		Clock100ms : BOOL;
		Clock200ms : BOOL;
		Clock500ms : BOOL;
		Clock1s : BOOL;
		Clock2s : BOOL;
		Drives_AllowLocalMode : BOOL;
		TestMode : BOOL; (** Bit to indicate test mode active*)
	END_STRUCT;
END_TYPE
```

### Standard.var
```iecst
VAR
	Std : Std_Vars;
END_VAR
```

### Program Logical/Standard/Standard/zzStd (IEC) - * Standard Functions

#### zzstd.var
```iecst
VAR
	TimerClkB : ARRAY[0..4] OF TON_10ms;
	TimerClkA : ARRAY[0..4] OF TON_10ms;
	n : UINT;
	TimerClkPT : ARRAY[0..4] OF UINT;
END_VAR
```

#### zzstd.ab
```automation-basic
;Version 1.00 First Issue
;Version 2.00 Added Bag[0] and Removed Mitsubishi M90xx's clock's
;Version 3.00 24/06/2009 New Bag 32bit etc.. D.J.

PROGRAM _INIT

END_PROGRAM

PROGRAM _CYCLIC

;Standard Clocks
TimerClkPT[0] = 5 	;100ms
TimerClkPT[1] = 10 	;200ms
TimerClkPT[2] = 25 	;500ms
TimerClkPT[3] = 50 	;1s
TimerClkPT[4] = 100 ;2s

LOOP n = 0 TO 4 DO

	TimerClkA[n].IN = NOT TimerClkB[n].Q
	TimerClkA[n].PT = TimerClkPT[n]
	TimerClkA[n] FUB TON_10ms()

	TimerClkB[n].IN = TimerClkA[n].Q
	TimerClkB[n].PT = TimerClkPT[n]
	TimerClkB[n] FUB TON_10ms()

ENDLOOP

Std.Clock100ms 	= TimerClkA[0].Q
Std.Clock200ms 	= TimerClkA[1].Q ;M9031
Std.Clock500ms 	= TimerClkA[2].Q
Std.Clock1s 	= TimerClkA[3].Q ;M9032
Std.Clock2s 	= TimerClkA[4].Q ;M9033
END_PROGRAM
```

### Hoist.var
```iecst
VAR
	OpcUa : {REDUND_UNREPLICABLE} OpcUa_type;
END_VAR
```

### Hoist.typ - Local data types
```iecst
TYPE
	OpcUa_type : 	STRUCT
		VC : ARRAY[230..254]OF OpcUa_VC_type;
	END_STRUCT;
	OpcUa_VC_type : 	STRUCT
		Read : OpcUa_VC_Read_type;
		Write : OpcUa_VC_Write_type;
	END_STRUCT;
	OpcUa_VC_Write_type : 	STRUCT
		Heartbeat : BOOL;
		PermissionToMove : BOOL;
		TargetPosition : USINT;
		ReleaseBag : BOOL;
		ReceiveBag : BOOL;
		LoadBag : BOOL;
		BagInTransit : BOOL;
	END_STRUCT;
	OpcUa_VC_Read_type : 	STRUCT
		StatusInfo : STRING[80];
		ActPosition : REAL;
		PositionNo : USINT;
		ReleaseBag : BOOL;
		ReceiveBag : BOOL;
		Heartbeat : BOOL;
		ReadyToReceive : BOOL;
		Auto : BOOL;
		Manual : BOOL;
		Error : BOOL;
		Weight : DINT;
		IsHome : BOOL;
		BagOnCarriage : BOOL;
		ChuteBlocked : BOOL;
	END_STRUCT;
END_TYPE
```

### Program Logical/Standard/HoistLibrary/HoistServer (IEC, version 2.00.1)

#### Main.st - Init, cyclic, exit code
```iecst
//V1.00.1  - TR - Add simulution mode.

PROGRAM _INIT

	selectedVC := 240;

END_PROGRAM

PROGRAM _CYCLIC

	MTBasicsPWM_0.DutyCycle		:= 50;
	MTBasicsPWM_0.Period		:= 2;
	MTBasicsPWM_0.Enable		:= TRUE;
	MTBasicsPWM_0(Enable:= TRUE,DutyCycle:= 50,Period:= 2,Update := 1);

	//FOR i := 38 TO 39 DO

pHmiOpcUa ACCESS ADR(OpcUa.VC[selectedVC]);

IF Std.TestMode THEN
		FOR i := 231 TO 254 DO

			hoist ACCESS ADR (OpcUa.VC[i]);

			hoist.Read.Heartbeat				:= MTBasicsPWM_0.Out; // NOT OpcUa.VC[i].Write.Heartbeat;
			hoist.Read.PositionNo 			:=	hoist.Write.TargetPosition;
			hoist.Read.Auto							:= 1;
			hoist.Read.ReadyToReceive 	:= 1;
			hoist.Read.IsHome						:= 1;

			ton_simulateRecv[i].IN 			:= 	hoist.Write.ReceiveBag;
			ton_simulateRecv[i].PT 			:= T#5s;
			ton_simulateRecv[i]();

			hoist.Read.ReceiveBag := ton_simulateRecv[i].Q;

			IF ton_simulateRecv[i].Q THEN
				hoist.Read.BagOnCarriage := 1;
			ELSIF hoist.Write.ReleaseBag THEN
				hoist.Read.BagOnCarriage := 0;
			END_IF;

		END_FOR;

ELSE
		FOR i := 231 TO 254 DO
			OpcUa.VC[i].Write.Heartbeat	:= MTBasicsPWM_0.Out; // NOT OpcUa.VC[i].Write.Heartbeat;
			//OpcUa.VC[i].Write.Heartbeat	:= pulse.Out;

			OpcUa.VC[i].Read.StatusInfo;
			OpcUa.VC[i].Read.ActPosition;
			OpcUa.VC[i].Read.PositionNo;
			OpcUa.VC[i].Read.ReceiveBag;
			OpcUa.VC[i].Read.ReleaseBag;
			OpcUa.VC[i].Read.Heartbeat;
			OpcUa.VC[i].Read.ReadyToReceive;

		END_FOR;

END_IF;

	(* Establish a connection to the client *)

(*	ReadHeartbeat;

	CASE Connect_to_OpcUaServer_step OF

		WAIT:

			IF Connect_OpcUa THEN

				Connect_to_OpcUaServer_step := CONNECT_TO_OPCUA;
			END_IF;

		CONNECT_TO_OPCUA:

			SessionConnectInfo_0.SecurityMsgMode := UASecurityMsgMode_None;
			SessionConnectInfo_0.SecurityPolicy := UASecurityPolicy_None;
			SessionConnectInfo_0.TransportProfile := UATP_UATcp;
			SessionConnectInfo_0.UserIdentityToken.UserIdentityTokenType := UAUITT_Anonymous;
			SessionConnectInfo_0.SessionTimeout := T#10m;
			SessionConnectInfo_0.MonitorConnection := T#10s;

			UA_Connect_0.ServerEndpointUrl := 'opc.tcp://10.44.10.244:4840';
			UA_Connect_0.Timeout := T#10s;
			UA_Connect_0.Execute := TRUE;
			UA_Connect_0.SessionConnectInfo := SessionConnectInfo_0;

			IF (UA_Connect_0.Done = 1) THEN
				UA_Connect_0.Execute := FALSE;
				Connect_OpcUa := FALSE;
				ConnectionHdl := UA_Connect_0.ConnectionHdl;
				Connect_to_OpcUaServer_step := GET_NAMESPACE;
			END_IF;

			IF (UA_Connect_0.Error = 1) THEN
				ConnectionHdl := 0;
				UA_Connect_0.Execute := FALSE;
				Connect_to_OpcUaServer_step := ERROR_OPCUA;
			END_IF;

		GET_NAMESPACE:

			UA_GetNamespaceIndex_0.ConnectionHdl := ConnectionHdl;
			UA_GetNamespaceIndex_0.NamespaceUri := 'urn:B&R/pv/';
			UA_GetNamespaceIndex_0.Timeout := T#5s;
			UA_GetNamespaceIndex_0.Execute := TRUE;

			IF (UA_GetNamespaceIndex_0.Done = 1) THEN
				NamespaceIndex := UA_GetNamespaceIndex_0.NamespaceIndex;
				UA_GetNamespaceIndex_0.Execute := FALSE;
				Connect_to_OpcUaServer_step := GET_NODE_HANDLE;
			END_IF;

			IF (UA_GetNamespaceIndex_0.Error = 1) THEN
				NamespaceIndex := 0;
				UA_GetNamespaceIndex_0.Execute := FALSE;
				Connect_to_OpcUaServer_step := ERROR_OPCUA;
			END_IF;

		GET_NODE_HANDLE:

			UANodeID_0[0].NamespaceIndex := NamespaceIndex;
			UANodeID_0[0].Identifier := '::Test_OpcUa_Client:WriteHeartbeat';
			UANodeID_0[0].IdentifierType := UAIdentifierType_String;

			UA_NodeGetHandleList_0.ConnectionHdl := ConnectionHdl;
			UA_NodeGetHandleList_0.NodeIDCount := 1;
			UA_NodeGetHandleList_0.NodeIDs := UANodeID_0;
			UA_NodeGetHandleList_0.Timeout := T#10s;
			UA_NodeGetHandleList_0.Execute := TRUE;

			IF (UA_NodeGetHandleList_0.Done = 1) THEN
				NodeHdls := UA_NodeGetHandleList_0.NodeHdls;
				UA_NodeGetHandleList_0.Execute := FALSE;
				Connect_to_OpcUaServer_step := READ_LIST;
			END_IF;

			IF (UA_NodeGetHandleList_0.Error = 1) THEN
				NodeHdls[0] := 0;

				UA_NodeGetHandleList_0.Execute := FALSE;
				Connect_to_OpcUaServer_step := ERROR_OPCUA;
			END_IF;

		READ_LIST:

			UANodeAdditionalInfo_0[0].AttributeId := UAAI_Value;
			UANodeAdditionalInfo_0[0].IndexRangeCount := 0;

			Variable_Rd0[0] := '::ServerTask:ReadHeartbeat';

			IF NOT UA_ReadList_0.Done THEN

				UA_ReadList_0
					(
					Execute := TRUE,
					ConnectionHdl := ConnectionHdl,
					NodeHdlCount := 1,
					NodeHdls := NodeHdls,
					NodeAddInfo := UANodeAdditionalInfo_0,
					Timeout := T#10s,
				Variables := Variable_Rd0);

				IF (UA_ReadList_0.Busy = 0) THEN
					UA_ReadList_0.Execute := FALSE;

					IF (UA_ReadList_0.Done = 1) THEN
						TimestampHeart := UA_ReadList_0.TimeStamps[0];

					END_IF;
					IF (UA_ReadList_0.Error = 1) THEN
						TimestampHeart := 0;
						Connect_to_OpcUaServer_step := ERROR_OPCUA;
					END_IF;
				END_IF;

			ELSIF StopReading THEN
				Connect_to_OpcUaServer_step := RELEASE_NODE;
				UA_ReadList_0.Execute := FALSE;

			ELSE
				UA_ReadList_0
					(
					Execute := FALSE,
					ConnectionHdl := ConnectionHdl,
					NodeHdlCount := 1,
					NodeHdls := NodeHdls,
					NodeAddInfo := UANodeAdditionalInfo_0,
					Timeout := T#10s,
				Variables := Variable_Rd0);
			END_IF;

		RELEASE_NODE:

			UA_NodeReleaseHandleList_0.ConnectionHdl := ConnectionHdl;
			UA_NodeReleaseHandleList_0.NodeHdlCount := 1;
			UA_NodeReleaseHandleList_0.NodeHdls := NodeHdls;
			UA_NodeReleaseHandleList_0.Timeout := T#10s;
			UA_NodeReleaseHandleList_0.Execute := TRUE;
			StopReading := FALSE;

			IF (UA_NodeReleaseHandleList_0.Done = 1) THEN
				NodeHdls[0] := 0;

				UA_NodeReleaseHandleList_0.Execute := FALSE;
				Connect_to_OpcUaServer_step := DISCONNECT_OPCUA;
			END_IF;

			IF (UA_NodeReleaseHandleList_0.Error = 1) THEN
				NodeHdls[0] := 0;

				UA_NodeReleaseHandleList_0.Execute := FALSE;
				Connect_to_OpcUaServer_step := ERROR_OPCUA;
			END_IF;

		DISCONNECT_OPCUA:

			UA_Disconnect_0.ConnectionHdl := ConnectionHdl;
			UA_Disconnect_0.Timeout := T#10s;
			UA_Disconnect_0.Execute := TRUE;

			IF (UA_Disconnect_0.Done = 1) THEN
				ConnectionHdl := 0;
				UA_Disconnect_0.Execute := FALSE;
				Connect_to_OpcUaServer_step := WAIT;
			END_IF;

			IF (UA_Disconnect_0.Error = 1) THEN
				ConnectionHdl := 0;
				UA_Disconnect_0.Execute := FALSE;
				Connect_to_OpcUaServer_step := ERROR_OPCUA;
			END_IF;

		ERROR_OPCUA:

	END_CASE;

	UA_Connect_0;
	UA_GetNamespaceIndex_0;
	UA_NodeGetHandleList_0;
	UA_NodeReleaseHandleList_0;
	UA_Disconnect_0;				*)

END_PROGRAM

PROGRAM _EXIT
	(* Insert code here *)

END_PROGRAM
```

#### Variables.var - Local variables
```iecst
(****************************************************)
VAR
	MTBasicsPWM_0 : MTBasicsPWM;
	i : USINT;
	pHmiOpcUa : REFERENCE TO OpcUa_VC_type;
	selectedVC : UINT;
	pulse : MTBasicsPWM;
	hoist : REFERENCE TO OpcUa_VC_type;
	ton_simulateRecv : ARRAY[230..255] OF TON;
END_VAR
```

- Fix IO Link Hardware file.docx (binary file, 12150 bytes)
- X20DS438A.hwx - *Version 1.1.0.0 (not shown)

- X20DS438A.hwx - *Version 1.9.1.0 (not shown)

### Fuse_Constants.var
```iecst
VAR CONSTANT
	MAX_FUSE_CHANNELS : USINT := 8; (*Max number of fuses in 1 bank*)
END_VAR
(*Reset Channels*)
VAR CONSTANT
	EB_SET_STATE_OFF : USINT := 1;
	EB_SET_STATE_ON : USINT := 2;
	EB_SET_STATE_RESET : USINT := 3;
END_VAR
```

### Fuse_Global.typ
```iecst
TYPE
	FuseSetting_typ : 	STRUCT
		GroupID : STRING[20]; (*Fuse Group Name*)
		MinVoltage : INT;
		MaxVoltage : INT;
		Channel : ARRAY[1..MAX_FUSE_CHANNELS]OF FuseChannelSetting_typ;
	END_STRUCT;
	FuseChannelSetting_typ : 	STRUCT
		FuseID : STRING[30]; (*Name can be to help identify the fuse*)
		SetState : USINT; (*State user wants to set the fuse too... Not Actual State*)
		TripCurrent : USINT;
	END_STRUCT;
END_TYPE
```

### Program Logical/Standard/IOLink/Fuses/FuseManagement (IEC, version 2.00.5)

#### Main.st - Init, cyclic, exit code
```iecst
//V1.00.0 -- First Release
//V1.00.1 -- Update so we monitor the status of the fuse and can send reset commands
//V1.00.2 -- Invert the fault lamp to a healthy lamp to stay consistent with hardwired devices
//V1.00.3 -- 03 March 2021. Improve error handling, on IO link fault

//V2.00.1 -- 19/03/2021  - Rewrite for better performance and add mappview hooks
//V2.00.2	-- Refactor as io link has a limit of 7 simultaneous function blocks
//V2.00.3	-- Refactor as io link has a limit of 7 simultaneous function blocks  Read/Write combined. not exclusive
//V2.00.4 -- Add visualization code so we can read out the live values.
//V2.00.5 -- Add front end visu

PROGRAM _INIT
	Fuse[1].pDevice := ADR('SL1.IF1.ST21.IF1.ST4.IF1');
	Fuse[2].pDevice := ADR('SL1.IF1.ST21.IF1.ST4.IF2');
	Fuse[3].pDevice := ADR('SL1.IF1.ST21.IF1.ST4.IF3');
	Fuse[4].pDevice := ADR('SL1.IF1.ST21.IF1.ST5.IF1');
	Fuse[5].pDevice := ADR('SL1.IF1.ST21.IF1.ST5.IF2');
	Fuse[6].pDevice := ADR('SL1.IF1.ST21.IF1.ST5.IF3');
	Fuse[7].pDevice := ADR('SL1.IF1.ST21.IF1.ST6.IF1');
	//
	Fuse[8].pDevice := ADR('SL1.IF1.ST22.IF1.ST4.IF1');
	Fuse[9].pDevice := ADR('SL1.IF1.ST22.IF1.ST4.IF2');
	Fuse[10].pDevice := ADR('SL1.IF1.ST22.IF1.ST4.IF3');
	Fuse[11].pDevice := ADR('SL1.IF1.ST22.IF1.ST5.IF1');
	//Fuse[12].pDevice := ADR('SL1.IF1.ST22.IF1.ST5.IF2');
	//Fuse[13].pDevice := ADR('SL1.IF1.ST22.IF1.ST5.IF3');

	gSettings.Fuse[1].GroupID := 'F71';
	gSettings.Fuse[2].GroupID := 'F72';
	gSettings.Fuse[3].GroupID := 'F81';
	gSettings.Fuse[4].GroupID := 'F73';
	gSettings.Fuse[5].GroupID := 'F74';
	gSettings.Fuse[6].GroupID := 'F75';
	gSettings.Fuse[7].GroupID := 'F76';
	//
	gSettings.Fuse[8].GroupID := 'F71';
	gSettings.Fuse[9].GroupID := 'F72';
	gSettings.Fuse[10].GroupID := 'F81';
	gSettings.Fuse[11].GroupID := 'F73';
	//gSettings.Fuse[12].GroupID := 'F73';
	//gSettings.Fuse[13].GroupID := 'F73';

	visu_index := 1;
	//alarm 	ACCESS ADR(Alarm[208]);
	FOR n := 1 TO MAX_FUSE_BANKS DO
		visu_settings ACCESS ADR(gSettings.Fuse[n]);
		IF (visu_settings.MinVoltage = 0) THEN visu_settings.MinVoltage := 1900; END_IF;
		IF (visu_settings.MaxVoltage = 0) THEN visu_settings.MaxVoltage := 2850; END_IF;
		FOR i := 1 TO MAX_FUSE_CHANNELS DO
			IF (visu_settings.Channel[i].TripCurrent = 0) THEN visu_settings.Channel[i].TripCurrent := 40; END_IF;
			IF (visu_settings.Channel[i].FuseID = '') THEN
				brsitoa(i,ADR(sIndex));
				visu_settings.Channel[i].FuseID := Fuse[n].Settings.GroupID;
				brsstrcat(ADR(visu_settings.Channel[i].FuseID),ADR('.'));
				brsstrcat(ADR(visu_settings.Channel[i].FuseID),ADR(sIndex));
			END_IF;
		END_FOR;
	END_FOR;
END_PROGRAM

PROGRAM _CYCLIC

	IF EDGEPOS(X[1005].X04) THEN
		reset[0] := 1;
	END_IF;
	IF EDGEPOS(X[2005].X04) THEN
		reset[1] := 1;
	END_IF;

	fuseFault[0] := 0;
	fuseFault[1] := 0;
	//alarm.On	:= 0;
	//alarm.Name	:= 0;

	//	IF visu_id <= MAX_FUSE_BANKS THEN
	//	visu_data ACCESS ADR(Fuse[visu_id]);
	//ELSE
	//	visu_data ACCESS ADR(Fuse[0]);
	//END_IF;

	FOR n := 1 TO MAX_FUSE_BANKS DO
		fuse ACCESS ADR(Fuse[n]);

		fuse.Settings := gSettings.Fuse[n];

		//Set up and monitoring of the fuses
		_config;
		// Monitor the state for messaging and alarms.
		IF fuse.Info.NoNodes > 0 THEN
			FOR i := 1 TO fuse.Info.NoNodes DO
				CASE fuse.Info.Channel[i].Status OF
					EB_STATE_NC: // Not connected

					EB_STATE_OFF:

					EB_STATE_ON:

					EB_STATE_TRIP:
						fuseFault[1] := 1;

					EB_STATE_I_90:

					EB_STATE_I_100:

					EB_STATE_TRIP_HARDWARE: // Fuse failed

					EB_STATE_TRIP_THERMAL:
						fuseFault[1] := 1;

					EB_STATE_TRIP_SW_OFF: // Turned off by hand

				END_CASE;
			END_FOR;
		END_IF;

	END_FOR;

	// Read live values when required.
	_visuRead;

	//Y[1006].Y10 := NOT fuseFault[0];
	//Y[2006].Y10 := NOT fuseFault[1];

END_PROGRAM
```
